KUKA KRL program: EPS_2_251112_SAMH03_A_20250918124115.src

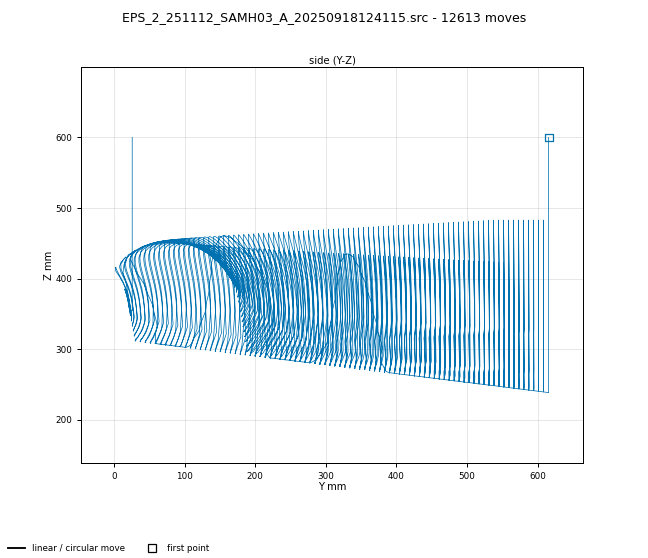
[picture p0: tool path of EPS_2_251112_SAMH03_A_20250918124115.src, 12613 of 12615 moves have a stored position in this frame; points joined in program order, loops and branches not executed]
&ACCESS RVP
&REL 4
&COMMENT QRS 19112012
&PARAM EDITMASK = *
DEF PART()
EXT BAS (BAS_COMMAND :IN,REAL :IN )
INT I
BAS (#INITMOV,0 )

;KUKA QRS Post kuka4.cps  Date:22-06-2017 !

File_ID=2847

QRS_PRE_INIT()

;Init var - Until changes are made in qrs_pre_init
Outlet_Square_prg=0
Inlet_1_Square_prg=0
Inlet_2_Square_prg=0
Inlet_3_Square_prg=0
Inlet_4_Square_prg=0
Inlet_5_Square_prg=0

Outlet_1={X 0.000, Y 541.230, Z 408.000, B 0.000, E1 0.000 }
Inlet_1={X 0.000, Y 545.490, Z 348.000, B 0.000, E1 229.000 }
Outlet_1_type=150
Inlet_1_type=150
;QRS#1=Sidecore dimensions
;QRS#2=150-6" PVC SDR 28
;QRS#3=150-6" PVC SDR 28
;QRS#4=
;QRS#5=
;QRS#6=
;QRS#7=
;QRS#8=
;QRS#9=10-06 PSX
;QRS#10=10-06 PSX
;QRS#11=
;QRS#12=
;QRS#13=
;QRS#14=
;QRS#15=
;QRS#16=1220x127x762 2,5'
;QRS#17=EPS Height
;QRS#18=483
;QRS#19=*
;QRS#20= UPDATED VERSION 22-06-2017
;QRS#21=*
Outlet_Square=070
Inlet_1_Square=070
Inlet_2_Square=0
Inlet_3_Square=0
Inlet_4_Square=0
Inlet_5_Square=0
Mill_Square=1
Outlet_Square_Prg=203
Inlet_1_Square_prg=203

QRS_INIT()

$ADVANCE=5

; T1
PTP {E1 173.598,E2 173.598}
PTP {X 0,Y 615.507,A -85,B 0,C 180,E1 173.598,E2 173.598,E3 0,E4 0,E5 0,E6 0}
QRS_SPEED_INIT()
LIN {X 0,Y 615.507,Z 600,A -85,B 0,C 180,E1 173.598,E2 173.598,E3 0,E4 0,E5 0,E6 0} C_VEL
LIN {X 0,Y 615.507,Z 248.674,A -85,B 0,C 180,E1 173.598,E2 173.598} C_VEL
LIN {X 0,Y 615.507,Z 240.494,A -85,B 0,C 180,E1 173.598,E2 173.598} C_VEL
LIN {X 0,Y 615.49,Z 238.494,A -85,B 0,C 180,E1 173.411,E2 173.411} C_VEL
LIN {X 0,Y 615.479,Z 238.505,A -85,B 0,C 180,E1 170.802,E2 170.802} C_VEL
LIN {X 0,Y 615.478,Z 238.506,A -85,B 0,C 180,E1 168.14,E2 168.14} C_VEL
LIN {X 0,Y 615.488,Z 238.494,A -85,B 0,C 180,E1 165.452,E2 165.452} C_VEL
LIN {X 0,Y 615.482,Z 238.506,A -85,B 0,C 180,E1 162.73,E2 162.73} C_VEL
LIN {X 0,Y 615.471,Z 238.504,A -85,B 0,C 180,E1 159.967,E2 159.967} C_VEL
LIN {X 0,Y 615.483,Z 238.497,A -85,B 0,C 180,E1 157.156,E2 157.156} C_VEL
LIN {X 0,Y 615.486,Z 238.51,A -85,B 0,C 180,E1 154.285,E2 154.285} C_VEL
LIN {X 0,Y 615.486,Z 238.495,A -85,B 0,C 180,E1 151.343,E2 151.343} C_VEL
LIN {X 0,Y 615.488,Z 238.51,A -85,B 0,C 180,E1 148.316,E2 148.316} C_VEL
LIN {X 0,Y 615.471,Z 238.504,A -85,B 0,C 180,E1 145.978,E2 145.978} C_VEL
LIN {X 0,Y 615.477,Z 238.497,A -85,B 0,C 180,E1 143.576,E2 143.576} C_VEL
LIN {X 0,Y 615.483,Z 238.501,A -85,B 0,C 180,E1 140.937,E2 140.937} C_VEL
LIN {X 0,Y 615.491,Z 238.511,A -85,B 0,C 180,E1 138.528,E2 138.528} C_VEL
LIN {X 0,Y 615.467,Z 238.502,A -85,B 0,C 180,E1 135.85,E2 135.85} C_VEL
LIN {X 0,Y 615.489,Z 238.497,A -85,B 0,C 180,E1 133.049,E2 133.049} C_VEL
LIN {X 0,Y 615.49,Z 238.508,A -85,B 0,C 180,E1 130.605,E2 130.605} C_VEL
LIN {X 0,Y 615.468,Z 238.506,A -85,B 0,C 180,E1 128.011,E2 128.011} C_VEL
LIN {X 0,Y 615.465,Z 238.5,A -85,B 0,C 180,E1 125.617,E2 125.617} C_VEL
LIN {X 0,Y 615.483,Z 238.496,A -85,B 0,C 180,E1 123.236,E2 123.236} C_VEL
LIN {X 0,Y 615.485,Z 238.5,A -85,B 0,C 180,E1 120.919,E2 120.919} C_VEL
LIN {X 0,Y 615.498,Z 238.512,A -85,B 0,C 180,E1 118.454,E2 118.454} C_VEL
LIN {X 0,Y 615.462,Z 238.502,A -85,B 0,C 180,E1 115.716,E2 115.716} C_VEL
LIN {X 0,Y 615.465,Z 238.5,A -85,B 0,C 180,E1 113.557,E2 113.557} C_VEL
LIN {X 0,Y 615.489,Z 238.504,A -85,B 0,C 180,E1 110.73,E2 110.73} C_VEL
LIN {X 0,Y 615.462,Z 238.506,A -85,B 0,C 180,E1 107.957,E2 107.957} C_VEL
LIN {X 0,Y 615.484,Z 238.496,A -85,B 0,C 180,E1 105.226,E2 105.226} C_VEL
LIN {X 0,Y 615.487,Z 238.511,A -85,B 0,C 180,E1 102.53,E2 102.53} C_VEL
LIN {X 0,Y 615.454,Z 238.506,A -85,B 0,C 180,E1 99.863,E2 99.863} C_VEL
LIN {X 0,Y 615.48,Z 238.497,A -85,B 0,C 180,E1 97.216,E2 97.216} C_VEL
LIN {X 0,Y 615.491,Z 238.509,A -85,B 0,C 180,E1 94.585,E2 94.585} C_VEL
LIN {X 0,Y 615.459,Z 238.507,A -85,B 0,C 180,E1 91.963,E2 91.963} C_VEL
LIN {X 0,Y 615.462,Z 238.5,A -85,B 0,C 180,E1 89.346,E2 89.346} C_VEL
LIN {X 0,Y 615.493,Z 238.503,A -85,B 0,C 180,E1 86.727,E2 86.727} C_VEL
LIN {X 0,Y 615.466,Z 238.509,A -85,B 0,C 180,E1 84.102,E2 84.102} C_VEL
LIN {X 0,Y 615.454,Z 238.502,A -85,B 0,C 180,E1 81.463,E2 81.463} C_VEL
LIN {X 0,Y 615.495,Z 238.5,A -85,B 0,C 180,E1 78.807,E2 78.807} C_VEL
LIN {X 0,Y 615.463,Z 238.509,A -85,B 0,C 180,E1 76.072,E2 76.072} C_VEL
LIN {X 0,Y 615.448,Z 238.504,A -85,B 0,C 180,E1 73.578,E2 73.578} C_VEL
LIN {X 0,Y 615.495,Z 238.505,A -85,B 0,C 180,E1 70.663,E2 70.663} C_VEL
LIN {X 0,Y 615.449,Z 238.507,A -85,B 0,C 180,E1 67.863,E2 67.863} C_VEL
LIN {X 0,Y 615.445,Z 238.506,A -85,B 0,C 180,E1 65.727,E2 65.727} C_VEL
LIN {X 0,Y 615.442,Z 238.505,A -85,B 0,C 180,E1 63.555,E2 63.555} C_VEL
LIN {X 0,Y 615.495,Z 238.507,A -85,B 0,C 180,E1 60.595,E2 60.595} C_VEL
LIN {X 0,Y 615.482,Z 238.513,A -85,B 0,C 180,E1 58.315,E2 58.315} C_VEL
LIN {X 0,Y 615.48,Z 238.537,A -85,B 0,C 180,E1 56.862,E2 56.862} C_VEL
LIN {X 0,Y 615.452,Z 250.671,A -85,B 0,C 180,E1 54.169,E2 54.169} C_VEL
LIN {X 0,Y 615.422,Z 260.877,A -85,B 0,C 180,E1 51.928,E2 51.928} C_VEL
LIN {X 0,Y 615.463,Z 264.848,A -85,B 0,C 180,E1 51.055,E2 51.055} C_VEL
LIN {X 0,Y 615.43,Z 339.353,A -85,B 0,C 180,E1 50.164,E2 50.164} C_VEL
LIN {X 0,Y 615.423,Z 347.654,A -85,B 0,C 180,E1 49.999,E2 49.999} C_VEL
LIN {X 0,Y 615.423,Z 357.187,A -85,B 0,C 180,E1 49.72,E2 49.72} C_VEL
LIN {X 0,Y 615.442,Z 365.491,A -85,B 0,C 180,E1 49.391,E2 49.391} C_VEL
LIN {X 0,Y 615.489,Z 373.933,A -85,B 0,C 180,E1 48.965,E2 48.965} C_VEL
LIN {X 0,Y 615.484,Z 382.137,A -85,B 0,C 180,E1 48.451,E2 48.451} C_VEL
LIN {X 0,Y 615.498,Z 390.744,A -85,B 0,C 180,E1 47.783,E2 47.783} C_VEL
LIN {X 0,Y 615.495,Z 399.09,A -85,B 0,C 180,E1 46.95,E2 46.95} C_VEL
LIN {X 0,Y 615.492,Z 405.175,A -85,B 0,C 180,E1 46.191,E2 46.191} C_VEL
LIN {X 0,Y 615.495,Z 409.938,A -85,B 0,C 180,E1 45.461,E2 45.461} C_VEL
LIN {X 0,Y 615.495,Z 412.871,A -85,B 0,C 180,E1 44.934,E2 44.934} C_VEL
LIN {X 0,Y 615.493,Z 416.877,A -85,B 0,C 180,E1 43.999,E2 43.999} C_VEL
LIN {X 0,Y 615.491,Z 419.769,A -85,B 0,C 180,E1 43.049,E2 43.049} C_VEL
LIN {X 0,Y 615.494,Z 421.587,A -85,B 0,C 180,E1 42.082,E2 42.082} C_VEL
LIN {X 0,Y 615.494,Z 422.345,A -85,B 0,C 180,E1 41.097,E2 41.097} C_VEL
LIN {X 0,Y 615.491,Z 421.957,A -85,B 0,C 180,E1 40.091,E2 40.091} C_VEL
LIN {X 0,Y 615.493,Z 419.87,A -85,B 0,C 180,E1 38.903,E2 38.903} C_VEL
LIN {X 0,Y 615.49,Z 417.42,A -85,B 0,C 180,E1 38.067,E2 38.067} C_VEL
LIN {X 0,Y 615.494,Z 414.081,A -85,B 0,C 180,E1 37.241,E2 37.241} C_VEL
LIN {X 0,Y 615.496,Z 409.786,A -85,B 0,C 180,E1 36.423,E2 36.423} C_VEL
LIN {X 0,Y 615.495,Z 404.427,A -85,B 0,C 180,E1 35.614,E2 35.614} C_VEL
LIN {X 0,Y 615.496,Z 396.778,A -85,B 0,C 180,E1 34.704,E2 34.704} C_VEL
LIN {X 0,Y 615.496,Z 389.446,A -85,B 0,C 180,E1 34.02,E2 34.02} C_VEL
LIN {X 0,Y 615.478,Z 382.157,A -85,B 0,C 180,E1 33.46,E2 33.46} C_VEL
LIN {X 0,Y 615.497,Z 373.88,A -85,B 0,C 180,E1 32.942,E2 32.942} C_VEL
LIN {X 0,Y 615.477,Z 365.174,A -85,B 0,C 180,E1 32.506,E2 32.506} C_VEL
LIN {X 0,Y 615.449,Z 356.53,A -85,B 0,C 180,E1 32.168,E2 32.168} C_VEL
LIN {X 0,Y 615.442,Z 346.706,A -85,B 0,C 180,E1 31.887,E2 31.887} C_VEL
LIN {X 0,Y 615.446,Z 335.604,A -85,B 0,C 180,E1 31.687,E2 31.687} C_VEL
LIN {X 0,Y 615.496,Z 264.804,A -85,B 0,C 180,E1 30.847,E2 30.847} C_VEL
LIN {X 0,Y 615.464,Z 252.68,A -85,B 0,C 180,E1 28.183,E2 28.183} C_VEL
LIN {X 0,Y 615.493,Z 240.882,A -85,B 0,C 180,E1 25.573,E2 25.573} C_VEL
LIN {X 0,Y 615.483,Z 238.5,A -85,B 0,C 180,E1 24.991,E2 24.991} C_VEL
LIN {X 0,Y 615.471,Z 238.501,A -85,B 0,C 180,E1 22.136,E2 22.136} C_VEL
LIN {X 0,Y 615.488,Z 238.509,A -85,B 0,C 180,E1 19.337,E2 19.337} C_VEL
LIN {X 0,Y 615.483,Z 238.495,A -85,B 0,C 180,E1 16.434,E2 16.434} C_VEL
LIN {X 0,Y 615.476,Z 238.505,A -85,B 0,C 180,E1 13.874,E2 13.874} C_VEL
LIN {X 0,Y 615.482,Z 238.506,A -85,B 0,C 180,E1 11.193,E2 11.193} C_VEL
LIN {X 0,Y 615.489,Z 238.494,A -85,B 0,C 180,E1 8.536,E2 8.536} C_VEL
LIN {X 0,Y 615.477,Z 238.505,A -85,B 0,C 180,E1 5.898,E2 5.898} C_VEL
LIN {X 0,Y 615.484,Z 238.508,A -85,B 0,C 180,E1 3.272,E2 3.272} C_VEL
LIN {X 0,Y 615.482,Z 238.496,A -85,B 0,C 180,E1 0.654,E2 0.654} C_VEL
LIN {X 0,Y 615.478,Z 238.501,A -85,B 0,C 180,E1 -1.964,E2 -1.964} C_VEL
LIN {X 0,Y 615.492,Z 238.511,A -85,B 0,C 180,E1 -4.585,E2 -4.585} C_VEL
LIN {X 0,Y 615.478,Z 238.498,A -85,B 0,C 180,E1 -7.216,E2 -7.216} C_VEL
LIN {X 0,Y 615.48,Z 238.499,A -85,B 0,C 180,E1 -9.863,E2 -9.863} C_VEL
LIN {X 0,Y 615.487,Z 238.514,A -85,B 0,C 180,E1 -12.531,E2 -12.531} C_VEL
LIN {X 0,Y 615.475,Z 238.499,A -85,B 0,C 180,E1 -15.227,E2 -15.227} C_VEL
LIN {X 0,Y 615.482,Z 238.5,A -85,B 0,C 180,E1 -17.957,E2 -17.957} C_VEL
LIN {X 0,Y 615.478,Z 238.509,A -85,B 0,C 180,E1 -20.731,E2 -20.731} C_VEL
LIN {X 0,Y 615.483,Z 238.495,A -85,B 0,C 180,E1 -23.557,E2 -23.557} C_VEL
LIN {X 0,Y 615.49,Z 238.513,A -85,B 0,C 180,E1 -26.444,E2 -26.444} C_VEL
LIN {X 0,Y 615.48,Z 238.511,A -85,B 0,C 180,E1 -28.659,E2 -28.659} C_VEL
LIN {X 0,Y 615.467,Z 238.502,A -85,B 0,C 180,E1 -31.085,E2 -31.085} C_VEL
LIN {X 0,Y 615.482,Z 238.496,A -85,B 0,C 180,E1 -33.535,E2 -33.535} C_VEL
LIN {X 0,Y 615.484,Z 238.514,A -85,B 0,C 180,E1 -36.425,E2 -36.425} C_VEL
LIN {X 0,Y 615.464,Z 238.503,A -85,B 0,C 180,E1 -39.061,E2 -39.061} C_VEL
LIN {X 0,Y 615.477,Z 238.497,A -85,B 0,C 180,E1 -41.475,E2 -41.475} C_VEL
LIN {X 0,Y 615.486,Z 238.504,A -85,B 0,C 180,E1 -44.15,E2 -44.15} C_VEL
LIN {X 0,Y 615.465,Z 238.505,A -85,B 0,C 180,E1 -46.955,E2 -46.955} C_VEL
LIN {X 0,Y 615.468,Z 238.499,A -85,B 0,C 180,E1 -49.393,E2 -49.393} C_VEL
LIN {X 0,Y 615.491,Z 238.499,A -85,B 0,C 180,E1 -51.988,E2 -51.988} C_VEL
LIN {X 0,Y 615.495,Z 238.51,A -85,B 0,C 180,E1 -54.386,E2 -54.386} C_VEL
LIN {X 0,Y 615.473,Z 238.509,A -85,B 0,C 180,E1 -56.764,E2 -56.764} C_VEL
LIN {X 0,Y 615.458,Z 238.505,A -85,B 0,C 180,E1 -59.08,E2 -59.08} C_VEL
LIN {X 0,Y 615.471,Z 238.498,A -85,B 0,C 180,E1 -61.553,E2 -61.553} C_VEL
LIN {X 0,Y 615.497,Z 238.511,A -85,B 0,C 180,E1 -64.429,E2 -64.429} C_VEL
LIN {X 0,Y 615.452,Z 238.505,A -85,B 0,C 180,E1 -67.155,E2 -67.155} C_VEL
LIN {X 0,Y 615.49,Z 238.596,A -85,B 0,C 180,E1 -67.839,E2 -67.839} C_VEL
LIN {X 0,Y 615.444,Z 257.739,A -85,B 0,C 180,E1 -70.661,E2 -70.661} C_VEL
LIN {X 0,Y 615.476,Z 276.68,A -85,B 0,C 180,E1 -73.414,E2 -73.414} C_VEL
LIN {X 0,Y 615.478,Z 296.787,A -85,B 0,C 180,E1 -76.294,E2 -76.294} C_VEL
LIN {X 0,Y 615.469,Z 315.645,A -85,B 0,C 180,E1 -78.966,E2 -78.966} C_VEL
LIN {X 0,Y 615.49,Z 322.035,A -85,B 0,C 180,E1 -79.868,E2 -79.868} C_VEL
LIN {X 0,Y 615.447,Z 399.978,A -85,B 0,C 180,E1 -80.801,E2 -80.801} C_VEL
LIN {X 0,Y 615.437,Z 409.726,A -85,B 0,C 180,E1 -81.008,E2 -81.008} C_VEL
LIN {X 0,Y 615.439,Z 420.178,A -85,B 0,C 180,E1 -81.339,E2 -81.339} C_VEL
LIN {X 0,Y 615.473,Z 430.438,A -85,B 0,C 180,E1 -81.794,E2 -81.794} C_VEL
LIN {X 0,Y 615.478,Z 440.206,A -85,B 0,C 180,E1 -82.372,E2 -82.372} C_VEL
LIN {X 0,Y 615.493,Z 447.938,A -85,B 0,C 180,E1 -82.942,E2 -82.942} C_VEL
LIN {X 0,Y 615.498,Z 455.337,A -85,B 0,C 180,E1 -83.608,E2 -83.608} C_VEL
LIN {X 0,Y 615.498,Z 462.739,A -85,B 0,C 180,E1 -84.431,E2 -84.431} C_VEL
LIN {X 0,Y 615.497,Z 468.534,A -85,B 0,C 180,E1 -85.252,E2 -85.252} C_VEL
LIN {X 0,Y 615.496,Z 473.101,A -85,B 0,C 180,E1 -86.072,E2 -86.072} C_VEL
LIN {X 0,Y 615.493,Z 476.069,A -85,B 0,C 180,E1 -86.727,E2 -86.727} C_VEL
LIN {X 0,Y 615.494,Z 478.357,A -85,B 0,C 180,E1 -87.382,E2 -87.382} C_VEL
LIN {X 0,Y 615.499,Z 480.085,A -85,B 0,C 180,E1 -88.037,E2 -88.037} C_VEL
LIN {X 0,Y 615.493,Z 481.33,A -85,B 0,C 180,E1 -88.692,E2 -88.692} C_VEL
LIN {X 0,Y 615.491,Z 482.104,A -85,B 0,C 180,E1 -89.346,E2 -89.346} C_VEL
LIN {X 0,Y 615.491,Z 482.389,A -85,B 0,C 180,E1 -90,E2 -90} C_VEL
LIN {X 0,Y 615.491,Z 482.104,A -85,B 0,C 180,E1 -90.654,E2 -90.654} C_VEL
LIN {X 0,Y 615.493,Z 481.33,A -85,B 0,C 180,E1 -91.309,E2 -91.309} C_VEL
LIN {X 0,Y 615.499,Z 480.085,A -85,B 0,C 180,E1 -91.963,E2 -91.963} C_VEL
LIN {X 0,Y 615.488,Z 477.22,A -85,B 0,C 180,E1 -92.945,E2 -92.945} C_VEL
LIN {X 0,Y 615.493,Z 474.602,A -85,B 0,C 180,E1 -93.601,E2 -93.601} C_VEL
LIN {X 0,Y 615.495,Z 469.482,A -85,B 0,C 180,E1 -94.585,E2 -94.585} C_VEL
LIN {X 0,Y 615.495,Z 463.968,A -85,B 0,C 180,E1 -95.405,E2 -95.405} C_VEL
LIN {X 0,Y 615.498,Z 457.017,A -85,B 0,C 180,E1 -96.227,E2 -96.227} C_VEL
LIN {X 0,Y 615.495,Z 449.859,A -85,B 0,C 180,E1 -96.901,E2 -96.901} C_VEL
LIN {X 0,Y 615.477,Z 442.624,A -85,B 0,C 180,E1 -97.463,E2 -97.463} C_VEL
LIN {X 0,Y 615.495,Z 434.868,A -85,B 0,C 180,E1 -97.958,E2 -97.958} C_VEL
LIN {X 0,Y 615.456,Z 426.924,A -85,B 0,C 180,E1 -98.372,E2 -98.372} C_VEL
LIN {X 0,Y 615.436,Z 417.772,A -85,B 0,C 180,E1 -98.744,E2 -98.744} C_VEL
LIN {X 0,Y 615.438,Z 409.713,A -85,B 0,C 180,E1 -98.992,E2 -98.992} C_VEL
LIN {X 0,Y 615.447,Z 399.958,A -85,B 0,C 180,E1 -99.199,E2 -99.199} C_VEL
LIN {X 0,Y 615.49,Z 322.033,A -85,B 0,C 180,E1 -100.132,E2 -100.132} C_VEL
LIN {X 0,Y 615.485,Z 302.697,A -85,B 0,C 180,E1 -102.865,E2 -102.865} C_VEL
LIN {X 0,Y 615.46,Z 283.779,A -85,B 0,C 180,E1 -105.566,E2 -105.566} C_VEL
LIN {X 0,Y 615.461,Z 263.931,A -85,B 0,C 180,E1 -108.434,E2 -108.434} C_VEL
LIN {X 0,Y 615.455,Z 247.068,A -85,B 0,C 180,E1 -110.907,E2 -110.907} C_VEL
LIN {X 0,Y 615.487,Z 238.497,A -85,B 0,C 180,E1 -112.187,E2 -112.187} C_VEL
LIN {X 0,Y 615.458,Z 238.506,A -85,B 0,C 180,E1 -114.993,E2 -114.993} C_VEL
LIN {X 0,Y 615.491,Z 238.501,A -85,B 0,C 180,E1 -117.914,E2 -117.914} C_VEL
LIN {X 0,Y 615.499,Z 238.494,A -85,B 0,C 180,E1 -120.159,E2 -120.159} C_VEL
LIN {X 0,Y 615.473,Z 238.498,A -85,B 0,C 180,E1 -122.458,E2 -122.458} C_VEL
LIN {X 0,Y 615.458,Z 238.503,A -85,B 0,C 180,E1 -124.816,E2 -124.816} C_VEL
LIN {X 0,Y 615.473,Z 238.509,A -85,B 0,C 180,E1 -127.243,E2 -127.243} C_VEL
LIN {X 0,Y 615.493,Z 238.497,A -85,B 0,C 180,E1 -130.089,E2 -130.089} C_VEL
LIN {X 0,Y 615.487,Z 238.495,A -85,B 0,C 180,E1 -132.352,E2 -132.352} C_VEL
LIN {X 0,Y 615.465,Z 238.506,A -85,B 0,C 180,E1 -135.07,E2 -135.07} C_VEL
LIN {X 0,Y 615.486,Z 238.502,A -85,B 0,C 180,E1 -137.919,E2 -137.919} C_VEL
LIN {X 0,Y 615.498,Z 238.493,A -85,B 0,C 180,E1 -140.25,E2 -140.25} C_VEL
LIN {X 0,Y 615.467,Z 238.505,A -85,B 0,C 180,E1 -143.065,E2 -143.065} C_VEL
LIN {X 0,Y 615.475,Z 238.51,A -85,B 0,C 180,E1 -145.3,E2 -145.3} C_VEL
LIN {X 0,Y 615.492,Z 238.509,A -85,B 0,C 180,E1 -147.667,E2 -147.667} C_VEL
LIN {X 0,Y 615.477,Z 238.497,A -85,B 0,C 180,E1 -150.593,E2 -150.593} C_VEL
LIN {X 0,Y 615.467,Z 238.503,A -85,B 0,C 180,E1 -152.957,E2 -152.957} C_VEL
LIN {X 0,Y 615.489,Z 238.508,A -85,B 0,C 180,E1 -155.728,E2 -155.728} C_VEL
LIN {X 0,Y 615.483,Z 238.495,A -85,B 0,C 180,E1 -158.568,E2 -158.568} C_VEL
LIN {X 0,Y 615.487,Z 238.51,A -85,B 0,C 180,E1 -161.393,E2 -161.393} C_VEL
LIN {X 0,Y 615.484,Z 238.499,A -85,B 0,C 180,E1 -164.094,E2 -164.094} C_VEL
LIN {X 0,Y 615.474,Z 238.499,A -85,B 0,C 180,E1 -166.798,E2 -166.798} C_VEL
LIN {X 0,Y 615.493,Z 238.512,A -85,B 0,C 180,E1 -169.473,E2 -169.473} C_VEL
LIN {X 0,Y 615.482,Z 238.499,A -85,B 0,C 180,E1 -172.124,E2 -172.124} C_VEL
LIN {X 0,Y 615.479,Z 238.497,A -85,B 0,C 180,E1 -174.758,E2 -174.758} C_VEL
LIN {X 0,Y 615.487,Z 238.509,A -85,B 0,C 180,E1 -177.382,E2 -177.382} C_VEL
LIN {X 0,Y 615.479,Z 238.503,A -85,B 0,C 180,E1 -179.999,E2 -179.999} C_VEL
LIN {X 0,Y 615.491,Z 238.493,A -85,B 0,C 180,E1 -182.617,E2 -182.617} C_VEL
LIN {X 0,Y 615.475,Z 238.507,A -85,B 0,C 180,E1 -185.241,E2 -185.241} C_VEL
LIN {X 0,Y 615.49,Z 238.494,A -85,B 0,C 180,E1 -186.589,E2 -186.589} C_VEL
LIN {X 0,Y 614.807,Z 238.652,A -85,B 0,C 180,E1 -187.135,E2 -187.135} C_VEL
LIN {X 0,Y 611.967,Z 239.065,A -85,B 0,C 180,E1 -188.021,E2 -188.021} C_VEL
LIN {X 0,Y 609.575,Z 239.378,A -85,B 0,C 180,E1 -188.733,E2 -188.733} C_VEL
LIN {X 0,Y 608.541,Z 239.496,A -85,B 0,C 180,E1 -189.283,E2 -189.283} C_VEL
LIN {X 0,Y 608.452,Z 239.505,A -85,B 0,C 180,E1 -189.469,E2 -189.469} C_VEL
LIN {X 0,Y 608.456,Z 239.503,A -85,B 0,C 180,E1 -191.999,E2 -191.999} C_VEL
LIN {X 0,Y 608.473,Z 239.497,A -85,B 0,C 180,E1 -194.72,E2 -194.72} C_VEL
LIN {X 0,Y 608.446,Z 239.51,A -85,B 0,C 180,E1 -197.476,E2 -197.476} C_VEL
LIN {X 0,Y 608.454,Z 239.5,A -85,B 0,C 180,E1 -200.274,E2 -200.274} C_VEL
LIN {X 0,Y 608.448,Z 239.5,A -85,B 0,C 180,E1 -202.476,E2 -202.476} C_VEL
LIN {X 0,Y 608.454,Z 239.506,A -85,B 0,C 180,E1 -205.3,E2 -205.3} C_VEL
LIN {X 0,Y 608.441,Z 239.512,A -85,B 0,C 180,E1 -207.517,E2 -207.517} C_VEL
LIN {X 0,Y 608.458,Z 239.503,A -85,B 0,C 180,E1 -209.972,E2 -209.972} C_VEL
LIN {X 0,Y 608.455,Z 239.499,A -85,B 0,C 180,E1 -212.523,E2 -212.523} C_VEL
LIN {X 0,Y 608.448,Z 239.506,A -85,B 0,C 180,E1 -215.276,E2 -215.276} C_VEL
LIN {X 0,Y 608.458,Z 239.506,A -85,B 0,C 180,E1 -217.746,E2 -217.746} C_VEL
LIN {X 0,Y 608.44,Z 239.502,A -85,B 0,C 180,E1 -220.329,E2 -220.329} C_VEL
LIN {X 0,Y 608.471,Z 239.504,A -85,B 0,C 180,E1 -223.31,E2 -223.31} C_VEL
LIN {X 0,Y 608.458,Z 239.501,A -85,B 0,C 180,E1 -226.13,E2 -226.13} C_VEL
LIN {X 0,Y 608.455,Z 239.5,A -85,B 0,C 180,E1 -228.824,E2 -228.824} C_VEL
LIN {X 0,Y 608.463,Z 239.506,A -85,B 0,C 180,E1 -231.412,E2 -231.412} C_VEL
LIN {X 0,Y 608.434,Z 239.506,A -85,B 0,C 180,E1 -233.954,E2 -233.954} C_VEL
LIN {X 0,Y 608.437,Z 239.502,A -85,B 0,C 180,E1 -236.328,E2 -236.328} C_VEL
LIN {X 0,Y 608.47,Z 239.498,A -85,B 0,C 180,E1 -238.727,E2 -238.727} C_VEL
LIN {X 0,Y 608.451,Z 239.508,A -85,B 0,C 180,E1 -241.734,E2 -241.734} C_VEL
LIN {X 0,Y 608.451,Z 239.501,A -85,B 0,C 180,E1 -244.281,E2 -244.281} C_VEL
LIN {X 0,Y 608.443,Z 239.502,A -85,B 0,C 180,E1 -246.876,E2 -246.876} C_VEL
LIN {X 0,Y 608.455,Z 239.507,A -85,B 0,C 180,E1 -249.726,E2 -249.726} C_VEL
LIN {X 0,Y 608.435,Z 239.508,A -85,B 0,C 180,E1 -251.828,E2 -251.828} C_VEL
LIN {X 0,Y 608.446,Z 239.505,A -85,B 0,C 180,E1 -253.906,E2 -253.906} C_VEL
LIN {X 0,Y 608.443,Z 239.505,A -85,B 0,C 180,E1 -255.988,E2 -255.988} C_VEL
LIN {X 0,Y 608.469,Z 239.498,A -85,B 0,C 180,E1 -258.676,E2 -258.676} C_VEL
LIN {X 0,Y 608.457,Z 239.506,A -85,B 0,C 180,E1 -261.364,E2 -261.364} C_VEL
LIN {X 0,Y 608.436,Z 239.505,A -85,B 0,C 180,E1 -264.033,E2 -264.033} C_VEL
LIN {X 0,Y 608.465,Z 239.498,A -85,B 0,C 180,E1 -266.689,E2 -266.689} C_VEL
LIN {X 0,Y 608.482,Z 239.502,A -85,B 0,C 180,E1 -269.338,E2 -269.338} C_VEL
LIN {X 0,Y 608.432,Z 239.506,A -85,B 0,C 180,E1 -271.986,E2 -271.986} C_VEL
LIN {X 0,Y 608.433,Z 239.506,A -85,B 0,C 180,E1 -273.974,E2 -273.974} C_VEL
LIN {X 0,Y 608.429,Z 239.503,A -85,B 0,C 180,E1 -276.633,E2 -276.633} C_VEL
LIN {X 0,Y 608.471,Z 239.503,A -85,B 0,C 180,E1 -279.305,E2 -279.305} C_VEL
LIN {X 0,Y 608.442,Z 239.505,A -85,B 0,C 180,E1 -282,E2 -282} C_VEL
LIN {X 0,Y 608.453,Z 239.5,A -85,B 0,C 180,E1 -284.721,E2 -284.721} C_VEL
LIN {X 0,Y 608.449,Z 239.509,A -85,B 0,C 180,E1 -287.476,E2 -287.476} C_VEL
LIN {X 0,Y 608.43,Z 239.503,A -85,B 0,C 180,E1 -290.275,E2 -290.275} C_VEL
LIN {X 0,Y 608.431,Z 239.502,A -85,B 0,C 180,E1 -292.473,E2 -292.473} C_VEL
LIN {X 0,Y 608.453,Z 239.505,A -85,B 0,C 180,E1 -295.3,E2 -295.3} C_VEL
LIN {X 0,Y 608.439,Z 239.511,A -85,B 0,C 180,E1 -297.518,E2 -297.518} C_VEL
LIN {X 0,Y 608.429,Z 239.507,A -85,B 0,C 180,E1 -299.967,E2 -299.967} C_VEL
LIN {X 0,Y 608.42,Z 239.504,A -85,B 0,C 180,E1 -302.518,E2 -302.518} C_VEL
LIN {X 0,Y 608.468,Z 239.719,A -85,B 0,C 180,E1 -303.174,E2 -303.174} C_VEL
LIN {X 0,Y 608.391,Z 252.562,A -85,B 0,C 180,E1 -306.04,E2 -306.04} C_VEL
LIN {X 0,Y 608.39,Z 262.483,A -85,B 0,C 180,E1 -308.233,E2 -308.233} C_VEL
LIN {X 0,Y 608.419,Z 265.192,A -85,B 0,C 180,E1 -308.829,E2 -308.829} C_VEL
LIN {X 0,Y 608.433,Z 340.315,A -85,B 0,C 180,E1 -309.737,E2 -309.737} C_VEL
LIN {X 0,Y 608.425,Z 350.261,A -85,B 0,C 180,E1 -309.953,E2 -309.953} C_VEL
LIN {X 0,Y 608.418,Z 361.668,A -85,B 0,C 180,E1 -310.327,E2 -310.327} C_VEL
LIN {X 0,Y 608.478,Z 372.532,A -85,B 0,C 180,E1 -310.844,E2 -310.844} C_VEL
LIN {X 0,Y 608.47,Z 380.777,A -85,B 0,C 180,E1 -311.345,E2 -311.345} C_VEL
LIN {X 0,Y 608.447,Z 387.854,A -85,B 0,C 180,E1 -311.867,E2 -311.867} C_VEL
LIN {X 0,Y 608.449,Z 394.437,A -85,B 0,C 180,E1 -312.45,E2 -312.45} C_VEL
LIN {X 0,Y 608.45,Z 400.823,A -85,B 0,C 180,E1 -313.132,E2 -313.132} C_VEL
LIN {X 0,Y 608.432,Z 406.518,A -85,B 0,C 180,E1 -313.871,E2 -313.871} C_VEL
LIN {X 0,Y 608.429,Z 412.234,A -85,B 0,C 180,E1 -314.797,E2 -314.797} C_VEL
LIN {X 0,Y 608.446,Z 416.628,A -85,B 0,C 180,E1 -315.736,E2 -315.736} C_VEL
LIN {X 0,Y 608.429,Z 419.796,A -85,B 0,C 180,E1 -316.694,E2 -316.694} C_VEL
LIN {X 0,Y 608.422,Z 422.239,A -85,B 0,C 180,E1 -317.937,E2 -317.937} C_VEL
LIN {X 0,Y 608.429,Z 422.92,A -85,B 0,C 180,E1 -318.823,E2 -318.823} C_VEL
LIN {X 0,Y 608.438,Z 422.718,A -85,B 0,C 180,E1 -319.697,E2 -319.697} C_VEL
LIN {X 0,Y 608.446,Z 421.437,A -85,B 0,C 180,E1 -320.704,E2 -320.704} C_VEL
LIN {X 0,Y 608.42,Z 418.688,A -85,B 0,C 180,E1 -321.764,E2 -321.764} C_VEL
LIN {X 0,Y 608.423,Z 415.661,A -85,B 0,C 180,E1 -322.575,E2 -322.575} C_VEL
LIN {X 0,Y 608.455,Z 411.045,A -85,B 0,C 180,E1 -323.499,E2 -323.499} C_VEL
LIN {X 0,Y 608.443,Z 407.033,A -85,B 0,C 180,E1 -324.146,E2 -324.146} C_VEL
LIN {X 0,Y 608.463,Z 400.994,A -85,B 0,C 180,E1 -324.938,E2 -324.938} C_VEL
LIN {X 0,Y 608.453,Z 394.527,A -85,B 0,C 180,E1 -325.631,E2 -325.631} C_VEL
LIN {X 0,Y 608.447,Z 386.559,A -85,B 0,C 180,E1 -326.329,E2 -326.329} C_VEL
LIN {X 0,Y 608.478,Z 376.473,A -85,B 0,C 180,E1 -327.024,E2 -327.024} C_VEL
LIN {X 0,Y 608.481,Z 366.615,A -85,B 0,C 180,E1 -327.542,E2 -327.542} C_VEL
LIN {X 0,Y 608.452,Z 357.646,A -85,B 0,C 180,E1 -327.906,E2 -327.906} C_VEL
LIN {X 0,Y 608.452,Z 348.309,A -85,B 0,C 180,E1 -328.186,E2 -328.186} C_VEL
LIN {X 0,Y 608.459,Z 339.339,A -85,B 0,C 180,E1 -328.369,E2 -328.369} C_VEL
LIN {X 0,Y 608.463,Z 265.177,A -85,B 0,C 180,E1 -329.264,E2 -329.264} C_VEL
LIN {X 0,Y 608.435,Z 252.294,A -85,B 0,C 180,E1 -332.108,E2 -332.108} C_VEL
LIN {X 0,Y 608.472,Z 239.5,A -85,B 0,C 180,E1 -334.975,E2 -334.975} C_VEL
LIN {X 0,Y 608.463,Z 239.498,A -85,B 0,C 180,E1 -337.595,E2 -337.595} C_VEL
LIN {X 0,Y 608.447,Z 239.51,A -85,B 0,C 180,E1 -340.43,E2 -340.43} C_VEL
LIN {X 0,Y 608.467,Z 239.498,A -85,B 0,C 180,E1 -343.467,E2 -343.467} C_VEL
LIN {X 0,Y 608.461,Z 239.501,A -85,B 0,C 180,E1 -345.981,E2 -345.981} C_VEL
LIN {X 0,Y 608.469,Z 239.505,A -85,B 0,C 180,E1 -348.677,E2 -348.677} C_VEL
LIN {X 0,Y 608.457,Z 239.499,A -85,B 0,C 180,E1 -351.365,E2 -351.365} C_VEL
LIN {X 0,Y 608.452,Z 239.503,A -85,B 0,C 180,E1 -354.034,E2 -354.034} C_VEL
LIN {X 0,Y 608.475,Z 239.504,A -85,B 0,C 180,E1 -356.69,E2 -356.69} C_VEL
LIN {X 0,Y 608.475,Z 239.497,A -85,B 0,C 180,E1 -359.339,E2 -359.339} C_VEL
LIN {X 0,Y 608.448,Z 239.503,A -85,B 0,C 180,E1 -361.986,E2 -361.986} C_VEL
LIN {X 0,Y 608.459,Z 239.507,A -85,B 0,C 180,E1 -364.638,E2 -364.638} C_VEL
LIN {X 0,Y 608.474,Z 239.497,A -85,B 0,C 180,E1 -367.3,E2 -367.3} C_VEL
LIN {X 0,Y 608.452,Z 239.502,A -85,B 0,C 180,E1 -369.978,E2 -369.978} C_VEL
LIN {X 0,Y 608.473,Z 239.505,A -85,B 0,C 180,E1 -372.677,E2 -372.677} C_VEL
LIN {X 0,Y 608.462,Z 239.498,A -85,B 0,C 180,E1 -375.407,E2 -375.407} C_VEL
LIN {X 0,Y 608.448,Z 239.505,A -85,B 0,C 180,E1 -378.172,E2 -378.172} C_VEL
LIN {X 0,Y 608.45,Z 239.503,A -85,B 0,C 180,E1 -380.982,E2 -380.982} C_VEL
LIN {X 0,Y 608.442,Z 239.502,A -85,B 0,C 180,E1 -383.125,E2 -383.125} C_VEL
LIN {X 0,Y 608.476,Z 239.497,A -85,B 0,C 180,E1 -385.724,E2 -385.724} C_VEL
LIN {X 0,Y 608.472,Z 239.506,A -85,B 0,C 180,E1 -388.622,E2 -388.622} C_VEL
LIN {X 0,Y 608.452,Z 239.5,A -85,B 0,C 180,E1 -391.318,E2 -391.318} C_VEL
LIN {X 0,Y 608.469,Z 239.498,A -85,B 0,C 180,E1 -393.736,E2 -393.736} C_VEL
LIN {X 0,Y 608.473,Z 239.501,A -85,B 0,C 180,E1 -396.091,E2 -396.091} C_VEL
LIN {X 0,Y 608.458,Z 239.508,A -85,B 0,C 180,E1 -398.589,E2 -398.589} C_VEL
LIN {X 0,Y 608.448,Z 239.5,A -85,B 0,C 180,E1 -401.342,E2 -401.342} C_VEL
LIN {X 0,Y 608.453,Z 239.506,A -85,B 0,C 180,E1 -404.265,E2 -404.265} C_VEL
LIN {X 0,Y 608.434,Z 239.504,A -85,B 0,C 180,E1 -407.04,E2 -407.04} C_VEL
LIN {X 0,Y 608.448,Z 239.501,A -85,B 0,C 180,E1 -409.698,E2 -409.698} C_VEL
LIN {X 0,Y 608.469,Z 239.504,A -85,B 0,C 180,E1 -412.255,E2 -412.255} C_VEL
LIN {X 0,Y 608.437,Z 239.508,A -85,B 0,C 180,E1 -414.723,E2 -414.723} C_VEL
LIN {X 0,Y 608.446,Z 239.502,A -85,B 0,C 180,E1 -417.121,E2 -417.121} C_VEL
LIN {X 0,Y 608.471,Z 239.501,A -85,B 0,C 180,E1 -420.028,E2 -420.028} C_VEL
LIN {X 0,Y 608.463,Z 239.504,A -85,B 0,C 180,E1 -422.796,E2 -422.796} C_VEL
LIN {X 0,Y 608.441,Z 239.501,A -85,B 0,C 180,E1 -425.429,E2 -425.429} C_VEL
LIN {X 0,Y 608.481,Z 239.663,A -85,B 0,C 180,E1 -427.73,E2 -427.73} C_VEL
LIN {X 0,Y 608.509,Z 256.575,A -85,B 0,C 180,E1 -430.256,E2 -430.256} C_VEL
LIN {X 0,Y 608.446,Z 274.378,A -85,B 0,C 180,E1 -432.87,E2 -432.87} C_VEL
LIN {X 0,Y 608.473,Z 292.18,A -85,B 0,C 180,E1 -435.451,E2 -435.451} C_VEL
LIN {X 0,Y 608.47,Z 311.169,A -85,B 0,C 180,E1 -438.17,E2 -438.17} C_VEL
LIN {X 0,Y 608.463,Z 322.296,A -85,B 0,C 180,E1 -439.75,E2 -439.75} C_VEL
LIN {X 0,Y 608.474,Z 400.465,A -85,B 0,C 180,E1 -440.695,E2 -440.695} C_VEL
LIN {X 0,Y 608.439,Z 410.088,A -85,B 0,C 180,E1 -440.904,E2 -440.904} C_VEL
LIN {X 0,Y 608.428,Z 421.626,A -85,B 0,C 180,E1 -441.28,E2 -441.28} C_VEL
LIN {X 0,Y 608.472,Z 432.238,A -85,B 0,C 180,E1 -441.783,E2 -441.783} C_VEL
LIN {X 0,Y 608.458,Z 440.546,A -85,B 0,C 180,E1 -442.284,E2 -442.284} C_VEL
LIN {X 0,Y 608.459,Z 448.404,A -85,B 0,C 180,E1 -442.868,E2 -442.868} C_VEL
LIN {X 0,Y 608.466,Z 455.358,A -85,B 0,C 180,E1 -443.496,E2 -443.496} C_VEL
LIN {X 0,Y 608.469,Z 463.193,A -85,B 0,C 180,E1 -444.366,E2 -444.366} C_VEL
LIN {X 0,Y 608.448,Z 469.028,A -85,B 0,C 180,E1 -445.197,E2 -445.197} C_VEL
LIN {X 0,Y 608.434,Z 473.632,A -85,B 0,C 180,E1 -446.026,E2 -446.026} C_VEL
LIN {X 0,Y 608.425,Z 476.622,A -85,B 0,C 180,E1 -446.689,E2 -446.689} C_VEL
LIN {X 0,Y 608.423,Z 478.932,A -85,B 0,C 180,E1 -447.352,E2 -447.352} C_VEL
LIN {X 0,Y 608.444,Z 480.679,A -85,B 0,C 180,E1 -448.014,E2 -448.014} C_VEL
LIN {X 0,Y 608.446,Z 481.934,A -85,B 0,C 180,E1 -448.676,E2 -448.676} C_VEL
LIN {X 0,Y 608.434,Z 482.714,A -85,B 0,C 180,E1 -449.338,E2 -449.338} C_VEL
LIN {X 0,Y 608.431,Z 483,A -85,B 0,C 180,E1 -450,E2 -450} C_VEL
LIN {X 0,Y 608.434,Z 482.714,A -85,B 0,C 180,E1 -450.662,E2 -450.662} C_VEL
LIN {X 0,Y 608.445,Z 481.933,A -85,B 0,C 180,E1 -451.324,E2 -451.324} C_VEL
LIN {X 0,Y 608.444,Z 480.678,A -85,B 0,C 180,E1 -451.986,E2 -451.986} C_VEL
LIN {X 0,Y 608.444,Z 477.785,A -85,B 0,C 180,E1 -452.98,E2 -452.98} C_VEL
LIN {X 0,Y 608.447,Z 475.146,A -85,B 0,C 180,E1 -453.642,E2 -453.642} C_VEL
LIN {X 0,Y 608.431,Z 469.984,A -85,B 0,C 180,E1 -454.638,E2 -454.638} C_VEL
LIN {X 0,Y 608.46,Z 464.429,A -85,B 0,C 180,E1 -455.468,E2 -455.468} C_VEL
LIN {X 0,Y 608.455,Z 456.67,A -85,B 0,C 180,E1 -456.376,E2 -456.376} C_VEL
LIN {X 0,Y 608.452,Z 449.414,A -85,B 0,C 180,E1 -457.049,E2 -457.049} C_VEL
LIN {X 0,Y 608.459,Z 441.76,A -85,B 0,C 180,E1 -457.633,E2 -457.633} C_VEL
LIN {X 0,Y 608.483,Z 433.719,A -85,B 0,C 180,E1 -458.134,E2 -458.134} C_VEL
LIN {X 0,Y 608.452,Z 425.389,A -85,B 0,C 180,E1 -458.552,E2 -458.552} C_VEL
LIN {X 0,Y 608.433,Z 416.888,A -85,B 0,C 180,E1 -458.887,E2 -458.887} C_VEL
LIN {X 0,Y 608.439,Z 407.585,A -85,B 0,C 180,E1 -459.16,E2 -459.16} C_VEL
LIN {X 0,Y 608.482,Z 396.548,A -85,B 0,C 180,E1 -459.368,E2 -459.368} C_VEL
LIN {X 0,Y 608.463,Z 322.293,A -85,B 0,C 180,E1 -460.25,E2 -460.25} C_VEL
LIN {X 0,Y 608.481,Z 301.672,A -85,B 0,C 180,E1 -463.186,E2 -463.186} C_VEL
LIN {X 0,Y 608.489,Z 281.496,A -85,B 0,C 180,E1 -466.093,E2 -466.093} C_VEL
LIN {X 0,Y 608.478,Z 262.507,A -85,B 0,C 180,E1 -468.869,E2 -468.869} C_VEL
LIN {X 0,Y 608.546,Z 244.704,A -85,B 0,C 180,E1 -471.51,E2 -471.51} C_VEL
LIN {X 0,Y 608.447,Z 239.502,A -85,B 0,C 180,E1 -472.317,E2 -472.317} C_VEL
LIN {X 0,Y 608.441,Z 239.501,A -85,B 0,C 180,E1 -474.571,E2 -474.571} C_VEL
LIN {X 0,Y 608.463,Z 239.504,A -85,B 0,C 180,E1 -477.204,E2 -477.204} C_VEL
LIN {X 0,Y 608.471,Z 239.501,A -85,B 0,C 180,E1 -479.972,E2 -479.972} C_VEL
LIN {X 0,Y 608.446,Z 239.502,A -85,B 0,C 180,E1 -482.88,E2 -482.88} C_VEL
LIN {X 0,Y 608.438,Z 239.508,A -85,B 0,C 180,E1 -485.277,E2 -485.277} C_VEL
LIN {X 0,Y 608.468,Z 239.498,A -85,B 0,C 180,E1 -488.24,E2 -488.24} C_VEL
LIN {X 0,Y 608.456,Z 239.507,A -85,B 0,C 180,E1 -491.341,E2 -491.341} C_VEL
LIN {X 0,Y 608.459,Z 239.499,A -85,B 0,C 180,E1 -494.264,E2 -494.264} C_VEL
LIN {X 0,Y 608.432,Z 239.505,A -85,B 0,C 180,E1 -497.038,E2 -497.038} C_VEL
LIN {X 0,Y 608.45,Z 239.508,A -85,B 0,C 180,E1 -499.696,E2 -499.696} C_VEL
LIN {X 0,Y 608.464,Z 239.499,A -85,B 0,C 180,E1 -502.253,E2 -502.253} C_VEL
LIN {X 0,Y 608.439,Z 239.502,A -85,B 0,C 180,E1 -504.722,E2 -504.722} C_VEL
LIN {X 0,Y 608.465,Z 239.508,A -85,B 0,C 180,E1 -507.476,E2 -507.476} C_VEL
LIN {X 0,Y 608.474,Z 239.498,A -85,B 0,C 180,E1 -510.221,E2 -510.221} C_VEL
LIN {X 0,Y 608.464,Z 239.499,A -85,B 0,C 180,E1 -512.794,E2 -512.794} C_VEL
LIN {X 0,Y 608.447,Z 239.509,A -85,B 0,C 180,E1 -515.428,E2 -515.428} C_VEL
LIN {X 0,Y 608.466,Z 239.498,A -85,B 0,C 180,E1 -518.308,E2 -518.308} C_VEL
LIN {X 0,Y 608.451,Z 239.504,A -85,B 0,C 180,E1 -521.13,E2 -521.13} C_VEL
LIN {X 0,Y 608.46,Z 239.503,A -85,B 0,C 180,E1 -523.906,E2 -523.906} C_VEL
LIN {X 0,Y 608.454,Z 239.499,A -85,B 0,C 180,E1 -526.643,E2 -526.643} C_VEL
LIN {X 0,Y 608.464,Z 239.506,A -85,B 0,C 180,E1 -529.35,E2 -529.35} C_VEL
LIN {X 0,Y 608.473,Z 239.5,A -85,B 0,C 180,E1 -532.033,E2 -532.033} C_VEL
LIN {X 0,Y 608.458,Z 239.499,A -85,B 0,C 180,E1 -534.698,E2 -534.698} C_VEL
LIN {X 0,Y 608.477,Z 239.504,A -85,B 0,C 180,E1 -537.351,E2 -537.351} C_VEL
LIN {X 0,Y 608.469,Z 239.501,A -85,B 0,C 180,E1 -539.999,E2 -539.999} C_VEL
LIN {X 0,Y 608.481,Z 239.496,A -85,B 0,C 180,E1 -542.647,E2 -542.647} C_VEL
LIN {X 0,Y 608.455,Z 239.506,A -85,B 0,C 180,E1 -545.301,E2 -545.301} C_VEL
LIN {X 0,Y 608.472,Z 239.501,A -85,B 0,C 180,E1 -547.966,E2 -547.966} C_VEL
LIN {X 0,Y 608.452,Z 239.505,A -85,B 0,C 180,E1 -549.469,E2 -549.469} C_VEL
LIN {X 0,Y 607.773,Z 239.588,A -85,B 0,C 180,E1 -550.022,E2 -550.022} C_VEL
LIN {X 0,Y 604.919,Z 239.941,A -85,B 0,C 180,E1 -550.919,E2 -550.919} C_VEL
LIN {X 0,Y 602.516,Z 240.248,A -85,B 0,C 180,E1 -551.64,E2 -551.64} C_VEL
LIN {X 0,Y 601.488,Z 240.369,A -85,B 0,C 180,E1 -552.197,E2 -552.197} C_VEL
LIN {X 0,Y 601.406,Z 240.378,A -85,B 0,C 180,E1 -552.385,E2 -552.385} C_VEL
LIN {X 0,Y 601.426,Z 240.376,A -85,B 0,C 180,E1 -554.896,E2 -554.896} C_VEL
LIN {X 0,Y 601.427,Z 240.377,A -85,B 0,C 180,E1 -556.985,E2 -556.985} C_VEL
LIN {X 0,Y 601.399,Z 240.384,A -85,B 0,C 180,E1 -559.809,E2 -559.809} C_VEL
LIN {X 0,Y 601.405,Z 240.377,A -85,B 0,C 180,E1 -562.605,E2 -562.605} C_VEL
LIN {X 0,Y 601.399,Z 240.379,A -85,B 0,C 180,E1 -564.878,E2 -564.878} C_VEL
LIN {X 0,Y 601.413,Z 240.382,A -85,B 0,C 180,E1 -567.867,E2 -567.867} C_VEL
LIN {X 0,Y 601.418,Z 240.378,A -85,B 0,C 180,E1 -570.164,E2 -570.164} C_VEL
LIN {X 0,Y 601.417,Z 240.376,A -85,B 0,C 180,E1 -572.716,E2 -572.716} C_VEL
LIN {X 0,Y 601.415,Z 240.38,A -85,B 0,C 180,E1 -575.116,E2 -575.116} C_VEL
LIN {X 0,Y 601.425,Z 240.383,A -85,B 0,C 180,E1 -577.419,E2 -577.419} C_VEL
LIN {X 0,Y 601.401,Z 240.382,A -85,B 0,C 180,E1 -579.995,E2 -579.995} C_VEL
LIN {X 0,Y 601.403,Z 240.378,A -85,B 0,C 180,E1 -582.67,E2 -582.67} C_VEL
LIN {X 0,Y 601.415,Z 240.386,A -85,B 0,C 180,E1 -585.482,E2 -585.482} C_VEL
LIN {X 0,Y 601.416,Z 240.376,A -85,B 0,C 180,E1 -588.406,E2 -588.406} C_VEL
LIN {X 0,Y 601.429,Z 240.376,A -85,B 0,C 180,E1 -590.876,E2 -590.876} C_VEL
LIN {X 0,Y 601.413,Z 240.384,A -85,B 0,C 180,E1 -593.736,E2 -593.736} C_VEL
LIN {X 0,Y 601.422,Z 240.378,A -85,B 0,C 180,E1 -596.064,E2 -596.064} C_VEL
LIN {X 0,Y 601.433,Z 240.374,A -85,B 0,C 180,E1 -598.541,E2 -598.541} C_VEL
LIN {X 0,Y 601.436,Z 240.381,A -85,B 0,C 180,E1 -601.374,E2 -601.374} C_VEL
LIN {X 0,Y 601.399,Z 240.388,A -85,B 0,C 180,E1 -603.636,E2 -603.636} C_VEL
LIN {X 0,Y 601.408,Z 240.377,A -85,B 0,C 180,E1 -606.59,E2 -606.59} C_VEL
LIN {X 0,Y 601.429,Z 240.384,A -85,B 0,C 180,E1 -609.478,E2 -609.478} C_VEL
LIN {X 0,Y 601.385,Z 240.381,A -85,B 0,C 180,E1 -612.311,E2 -612.311} C_VEL
LIN {X 0,Y 601.404,Z 240.378,A -85,B 0,C 180,E1 -614.409,E2 -614.409} C_VEL
LIN {X 0,Y 601.418,Z 240.38,A -85,B 0,C 180,E1 -617.172,E2 -617.172} C_VEL
LIN {X 0,Y 601.416,Z 240.381,A -85,B 0,C 180,E1 -619.905,E2 -619.905} C_VEL
LIN {X 0,Y 601.431,Z 240.374,A -85,B 0,C 180,E1 -622.615,E2 -622.615} C_VEL
LIN {X 0,Y 601.424,Z 240.381,A -85,B 0,C 180,E1 -625.308,E2 -625.308} C_VEL
LIN {X 0,Y 601.403,Z 240.382,A -85,B 0,C 180,E1 -627.991,E2 -627.991} C_VEL
LIN {X 0,Y 601.431,Z 240.374,A -85,B 0,C 180,E1 -630.669,E2 -630.669} C_VEL
LIN {X 0,Y 601.433,Z 240.381,A -85,B 0,C 180,E1 -633.349,E2 -633.349} C_VEL
LIN {X 0,Y 601.39,Z 240.383,A -85,B 0,C 180,E1 -636.037,E2 -636.037} C_VEL
LIN {X 0,Y 601.422,Z 240.378,A -85,B 0,C 180,E1 -638.061,E2 -638.061} C_VEL
LIN {X 0,Y 601.412,Z 240.379,A -85,B 0,C 180,E1 -641.011,E2 -641.011} C_VEL
LIN {X 0,Y 601.41,Z 240.387,A -85,B 0,C 180,E1 -643.516,E2 -643.516} C_VEL
LIN {X 0,Y 601.412,Z 240.378,A -85,B 0,C 180,E1 -646.287,E2 -646.287} C_VEL
LIN {X 0,Y 601.406,Z 240.38,A -85,B 0,C 180,E1 -649.099,E2 -649.099} C_VEL
LIN {X 0,Y 601.389,Z 240.384,A -85,B 0,C 180,E1 -651.959,E2 -651.959} C_VEL
LIN {X 0,Y 601.391,Z 240.38,A -85,B 0,C 180,E1 -654.286,E2 -654.286} C_VEL
LIN {X 0,Y 601.446,Z 240.375,A -85,B 0,C 180,E1 -657.111,E2 -657.111} C_VEL
LIN {X 0,Y 601.407,Z 240.385,A -85,B 0,C 180,E1 -659.393,E2 -659.393} C_VEL
LIN {X 0,Y 601.394,Z 240.388,A -85,B 0,C 180,E1 -661.726,E2 -661.726} C_VEL
LIN {X 0,Y 601.424,Z 240.438,A -85,B 0,C 180,E1 -663.147,E2 -663.147} C_VEL
LIN {X 0,Y 601.323,Z 253.095,A -85,B 0,C 180,E1 -666.004,E2 -666.004} C_VEL
LIN {X 0,Y 601.344,Z 265.185,A -85,B 0,C 180,E1 -668.706,E2 -668.706} C_VEL
LIN {X 0,Y 601.483,Z 318.398,A -85,B 0,C 180,E1 -669.348,E2 -669.348} C_VEL
LIN {X 0,Y 601.448,Z 341.407,A -85,B 0,C 180,E1 -669.645,E2 -669.645} C_VEL
LIN {X 0,Y 601.418,Z 353.124,A -85,B 0,C 180,E1 -669.922,E2 -669.922} C_VEL
LIN {X 0,Y 601.414,Z 363.541,A -85,B 0,C 180,E1 -670.307,E2 -670.307} C_VEL
LIN {X 0,Y 601.438,Z 371.576,A -85,B 0,C 180,E1 -670.693,E2 -670.693} C_VEL
LIN {X 0,Y 601.419,Z 380.088,A -85,B 0,C 180,E1 -671.206,E2 -671.206} C_VEL
LIN {X 0,Y 601.393,Z 387.664,A -85,B 0,C 180,E1 -671.767,E2 -671.767} C_VEL
LIN {X 0,Y 601.373,Z 394.744,A -85,B 0,C 180,E1 -672.403,E2 -672.403} C_VEL
LIN {X 0,Y 601.374,Z 401.299,A -85,B 0,C 180,E1 -673.119,E2 -673.119} C_VEL
LIN {X 0,Y 601.361,Z 408.221,A -85,B 0,C 180,E1 -674.055,E2 -674.055} C_VEL
LIN {X 0,Y 601.366,Z 413.552,A -85,B 0,C 180,E1 -675.007,E2 -675.007} C_VEL
LIN {X 0,Y 601.362,Z 417.495,A -85,B 0,C 180,E1 -675.945,E2 -675.945} C_VEL
LIN {X 0,Y 601.331,Z 420.31,A -85,B 0,C 180,E1 -676.881,E2 -676.881} C_VEL
LIN {X 0,Y 601.335,Z 421.52,A -85,B 0,C 180,E1 -677.416,E2 -677.416} C_VEL
LIN {X 0,Y 601.32,Z 422.733,A -85,B 0,C 180,E1 -678.417,E2 -678.417} C_VEL
LIN {X 0,Y 601.308,Z 422.842,A -85,B 0,C 180,E1 -679.437,E2 -679.437} C_VEL
LIN {X 0,Y 601.321,Z 421.805,A -85,B 0,C 180,E1 -680.476,E2 -680.476} C_VEL
LIN {X 0,Y 601.319,Z 419.506,A -85,B 0,C 180,E1 -681.541,E2 -681.541} C_VEL
LIN {X 0,Y 601.353,Z 415.616,A -85,B 0,C 180,E1 -682.626,E2 -682.626} C_VEL
LIN {X 0,Y 601.358,Z 411.824,A -85,B 0,C 180,E1 -683.415,E2 -683.415} C_VEL
LIN {X 0,Y 601.353,Z 406.767,A -85,B 0,C 180,E1 -684.244,E2 -684.244} C_VEL
LIN {X 0,Y 601.377,Z 400.492,A -85,B 0,C 180,E1 -685.067,E2 -685.067} C_VEL
LIN {X 0,Y 601.407,Z 392.78,A -85,B 0,C 180,E1 -685.881,E2 -685.881} C_VEL
LIN {X 0,Y 601.407,Z 384.386,A -85,B 0,C 180,E1 -686.586,E2 -686.586} C_VEL
LIN {X 0,Y 601.464,Z 375.112,A -85,B 0,C 180,E1 -687.196,E2 -687.196} C_VEL
LIN {X 0,Y 601.442,Z 366.776,A -85,B 0,C 180,E1 -687.635,E2 -687.635} C_VEL
LIN {X 0,Y 601.444,Z 358.469,A -85,B 0,C 180,E1 -687.981,E2 -687.981} C_VEL
LIN {X 0,Y 601.427,Z 349.022,A -85,B 0,C 180,E1 -688.276,E2 -688.276} C_VEL
LIN {X 0,Y 601.478,Z 339.364,A -85,B 0,C 180,E1 -688.478,E2 -688.478} C_VEL
LIN {X 0,Y 601.4,Z 265.296,A -85,B 0,C 180,E1 -689.374,E2 -689.374} C_VEL
LIN {X 0,Y 601.379,Z 252.886,A -85,B 0,C 180,E1 -692.131,E2 -692.131} C_VEL
LIN {X 0,Y 601.411,Z 240.38,A -85,B 0,C 180,E1 -694.984,E2 -694.984} C_VEL
LIN {X 0,Y 601.404,Z 240.378,A -85,B 0,C 180,E1 -697.394,E2 -697.394} C_VEL
LIN {X 0,Y 601.4,Z 240.384,A -85,B 0,C 180,E1 -700.191,E2 -700.191} C_VEL
LIN {X 0,Y 601.427,Z 240.378,A -85,B 0,C 180,E1 -703.015,E2 -703.015} C_VEL
LIN {X 0,Y 601.41,Z 240.379,A -85,B 0,C 180,E1 -705.908,E2 -705.908} C_VEL
LIN {X 0,Y 601.426,Z 240.385,A -85,B 0,C 180,E1 -708.542,E2 -708.542} C_VEL
LIN {X 0,Y 601.435,Z 240.375,A -85,B 0,C 180,E1 -711.263,E2 -711.263} C_VEL
LIN {X 0,Y 601.405,Z 240.38,A -85,B 0,C 180,E1 -713.963,E2 -713.963} C_VEL
LIN {X 0,Y 601.426,Z 240.383,A -85,B 0,C 180,E1 -716.651,E2 -716.651} C_VEL
LIN {X 0,Y 601.446,Z 240.373,A -85,B 0,C 180,E1 -719.331,E2 -719.331} C_VEL
LIN {X 0,Y 601.418,Z 240.379,A -85,B 0,C 180,E1 -722.01,E2 -722.01} C_VEL
LIN {X 0,Y 601.426,Z 240.382,A -85,B 0,C 180,E1 -724.692,E2 -724.692} C_VEL
LIN {X 0,Y 601.444,Z 240.373,A -85,B 0,C 180,E1 -727.386,E2 -727.386} C_VEL
LIN {X 0,Y 601.429,Z 240.379,A -85,B 0,C 180,E1 -730.096,E2 -730.096} C_VEL
LIN {X 0,Y 601.416,Z 240.381,A -85,B 0,C 180,E1 -732.829,E2 -732.829} C_VEL
LIN {X 0,Y 601.407,Z 240.377,A -85,B 0,C 180,E1 -735.592,E2 -735.592} C_VEL
LIN {X 0,Y 601.419,Z 240.385,A -85,B 0,C 180,E1 -738.392,E2 -738.392} C_VEL
LIN {X 0,Y 601.402,Z 240.378,A -85,B 0,C 180,E1 -741.24,E2 -741.24} C_VEL
LIN {X 0,Y 601.454,Z 240.376,A -85,B 0,C 180,E1 -744.141,E2 -744.141} C_VEL
LIN {X 0,Y 601.438,Z 240.375,A -85,B 0,C 180,E1 -747.112,E2 -747.112} C_VEL
LIN {X 0,Y 601.418,Z 240.376,A -85,B 0,C 180,E1 -749.393,E2 -749.393} C_VEL
LIN {X 0,Y 601.404,Z 240.378,A -85,B 0,C 180,E1 -751.727,E2 -751.727} C_VEL
LIN {X 0,Y 601.425,Z 240.379,A -85,B 0,C 180,E1 -754.119,E2 -754.119} C_VEL
LIN {X 0,Y 601.402,Z 240.387,A -85,B 0,C 180,E1 -756.583,E2 -756.583} C_VEL
LIN {X 0,Y 601.436,Z 240.374,A -85,B 0,C 180,E1 -759.537,E2 -759.537} C_VEL
LIN {X 0,Y 601.406,Z 240.386,A -85,B 0,C 180,E1 -762.592,E2 -762.592} C_VEL
LIN {X 0,Y 601.421,Z 240.376,A -85,B 0,C 180,E1 -765.483,E2 -765.483} C_VEL
LIN {X 0,Y 601.422,Z 240.385,A -85,B 0,C 180,E1 -768.407,E2 -768.407} C_VEL
LIN {X 0,Y 601.427,Z 240.375,A -85,B 0,C 180,E1 -771.53,E2 -771.53} C_VEL
LIN {X 0,Y 601.403,Z 240.384,A -85,B 0,C 180,E1 -774.247,E2 -774.247} C_VEL
LIN {X 0,Y 601.427,Z 240.382,A -85,B 0,C 180,E1 -776.687,E2 -776.687} C_VEL
LIN {X 0,Y 601.407,Z 240.379,A -85,B 0,C 180,E1 -779.058,E2 -779.058} C_VEL
LIN {X 0,Y 601.414,Z 240.377,A -85,B 0,C 180,E1 -781.373,E2 -781.373} C_VEL
LIN {X 0,Y 601.414,Z 240.381,A -85,B 0,C 180,E1 -784.133,E2 -784.133} C_VEL
LIN {X 0,Y 601.413,Z 240.387,A -85,B 0,C 180,E1 -786.59,E2 -786.59} C_VEL
LIN {X 0,Y 601.412,Z 240.489,A -85,B 0,C 180,E1 -787.58,E2 -787.58} C_VEL
LIN {X 0,Y 601.607,Z 245.894,A -85,B 0,C 180,E1 -788.409,E2 -788.409} C_VEL
LIN {X 0,Y 601.505,Z 262.509,A -85,B 0,C 180,E1 -790.905,E2 -790.905} C_VEL
LIN {X 0,Y 601.515,Z 281.498,A -85,B 0,C 180,E1 -793.716,E2 -793.716} C_VEL
LIN {X 0,Y 601.43,Z 301.675,A -85,B 0,C 180,E1 -796.657,E2 -796.657} C_VEL
LIN {X 0,Y 601.372,Z 319.477,A -85,B 0,C 180,E1 -799.223,E2 -799.223} C_VEL
LIN {X 0,Y 601.389,Z 322.296,A -85,B 0,C 180,E1 -799.628,E2 -799.628} C_VEL
LIN {X 0,Y 601.469,Z 400.464,A -85,B 0,C 180,E1 -800.585,E2 -800.585} C_VEL
LIN {X 0,Y 601.432,Z 410.918,A -85,B 0,C 180,E1 -800.818,E2 -800.818} C_VEL
LIN {X 0,Y 601.414,Z 423.544,A -85,B 0,C 180,E1 -801.262,E2 -801.262} C_VEL
LIN {X 0,Y 601.437,Z 432.241,A -85,B 0,C 180,E1 -801.686,E2 -801.686} C_VEL
LIN {X 0,Y 601.402,Z 440.548,A -85,B 0,C 180,E1 -802.193,E2 -802.193} C_VEL
LIN {X 0,Y 601.409,Z 448.405,A -85,B 0,C 180,E1 -802.784,E2 -802.784} C_VEL
LIN {X 0,Y 601.412,Z 455.599,A -85,B 0,C 180,E1 -803.443,E2 -803.443} C_VEL
LIN {X 0,Y 601.391,Z 463.193,A -85,B 0,C 180,E1 -804.3,E2 -804.3} C_VEL
LIN {X 0,Y 601.38,Z 469.029,A -85,B 0,C 180,E1 -805.14,E2 -805.14} C_VEL
LIN {X 0,Y 601.345,Z 473.632,A -85,B 0,C 180,E1 -805.979,E2 -805.979} C_VEL
LIN {X 0,Y 601.344,Z 476.622,A -85,B 0,C 180,E1 -806.65,E2 -806.65} C_VEL
LIN {X 0,Y 601.326,Z 478.932,A -85,B 0,C 180,E1 -807.321,E2 -807.321} C_VEL
LIN {X 0,Y 601.343,Z 480.679,A -85,B 0,C 180,E1 -807.991,E2 -807.991} C_VEL
LIN {X 0,Y 601.345,Z 481.935,A -85,B 0,C 180,E1 -808.661,E2 -808.661} C_VEL
LIN {X 0,Y 601.335,Z 482.713,A -85,B 0,C 180,E1 -809.331,E2 -809.331} C_VEL
LIN {X 0,Y 601.332,Z 483,A -85,B 0,C 180,E1 -810,E2 -810} C_VEL
LIN {X 0,Y 601.335,Z 482.713,A -85,B 0,C 180,E1 -810.67,E2 -810.67} C_VEL
LIN {X 0,Y 601.345,Z 481.934,A -85,B 0,C 180,E1 -811.34,E2 -811.34} C_VEL
LIN {X 0,Y 601.343,Z 480.678,A -85,B 0,C 180,E1 -812.009,E2 -812.009} C_VEL
LIN {X 0,Y 601.343,Z 477.786,A -85,B 0,C 180,E1 -813.015,E2 -813.015} C_VEL
LIN {X 0,Y 601.365,Z 475.146,A -85,B 0,C 180,E1 -813.685,E2 -813.685} C_VEL
LIN {X 0,Y 601.341,Z 469.984,A -85,B 0,C 180,E1 -814.693,E2 -814.693} C_VEL
LIN {X 0,Y 601.383,Z 464.429,A -85,B 0,C 180,E1 -815.533,E2 -815.533} C_VEL
LIN {X 0,Y 601.394,Z 457.153,A -85,B 0,C 180,E1 -816.403,E2 -816.403} C_VEL
LIN {X 0,Y 601.413,Z 449.416,A -85,B 0,C 180,E1 -817.132,E2 -817.132} C_VEL
LIN {X 0,Y 601.424,Z 441.762,A -85,B 0,C 180,E1 -817.723,E2 -817.723} C_VEL
LIN {X 0,Y 601.445,Z 433.722,A -85,B 0,C 180,E1 -818.23,E2 -818.23} C_VEL
LIN {X 0,Y 601.428,Z 425.392,A -85,B 0,C 180,E1 -818.653,E2 -818.653} C_VEL
LIN {X 0,Y 601.423,Z 416.89,A -85,B 0,C 180,E1 -818.992,E2 -818.992} C_VEL
LIN {X 0,Y 601.451,Z 406.755,A -85,B 0,C 180,E1 -819.288,E2 -819.288} C_VEL
LIN {X 0,Y 601.485,Z 395.06,A -85,B 0,C 180,E1 -819.5,E2 -819.5} C_VEL
LIN {X 0,Y 601.389,Z 322.293,A -85,B 0,C 180,E1 -820.372,E2 -820.372} C_VEL
LIN {X 0,Y 601.46,Z 302.859,A -85,B 0,C 180,E1 -823.171,E2 -823.171} C_VEL
LIN {X 0,Y 601.475,Z 282.683,A -85,B 0,C 180,E1 -826.111,E2 -826.111} C_VEL
LIN {X 0,Y 601.507,Z 264.197,A -85,B 0,C 180,E1 -828.844,E2 -828.844} C_VEL
LIN {X 0,Y 601.589,Z 247.078,A -85,B 0,C 180,E1 -831.412,E2 -831.412} C_VEL
LIN {X 0,Y 601.557,Z 241.191,A -85,B 0,C 180,E1 -832.307,E2 -832.307} C_VEL
LIN {X 0,Y 601.436,Z 240.378,A -85,B 0,C 180,E1 -832.473,E2 -832.473} C_VEL
LIN {X 0,Y 601.394,Z 240.381,A -85,B 0,C 180,E1 -834.879,E2 -834.879} C_VEL
LIN {X 0,Y 601.406,Z 240.386,A -85,B 0,C 180,E1 -837.361,E2 -837.361} C_VEL
LIN {X 0,Y 601.428,Z 240.376,A -85,B 0,C 180,E1 -840.164,E2 -840.164} C_VEL
LIN {X 0,Y 601.412,Z 240.377,A -85,B 0,C 180,E1 -842.714,E2 -842.714} C_VEL
LIN {X 0,Y 601.385,Z 240.384,A -85,B 0,C 180,E1 -845.11,E2 -845.11} C_VEL
LIN {X 0,Y 601.431,Z 240.383,A -85,B 0,C 180,E1 -847.419,E2 -847.419} C_VEL
LIN {X 0,Y 601.399,Z 240.381,A -85,B 0,C 180,E1 -849.995,E2 -849.995} C_VEL
LIN {X 0,Y 601.405,Z 240.378,A -85,B 0,C 180,E1 -852.67,E2 -852.67} C_VEL
LIN {X 0,Y 601.423,Z 240.386,A -85,B 0,C 180,E1 -855.482,E2 -855.482} C_VEL
LIN {X 0,Y 601.416,Z 240.376,A -85,B 0,C 180,E1 -858.407,E2 -858.407} C_VEL
LIN {X 0,Y 601.405,Z 240.379,A -85,B 0,C 180,E1 -860.873,E2 -860.873} C_VEL
LIN {X 0,Y 601.439,Z 240.38,A -85,B 0,C 180,E1 -863.733,E2 -863.733} C_VEL
LIN {X 0,Y 601.422,Z 240.376,A -85,B 0,C 180,E1 -866.686,E2 -866.686} C_VEL
LIN {X 0,Y 601.406,Z 240.38,A -85,B 0,C 180,E1 -869.057,E2 -869.057} C_VEL
LIN {X 0,Y 601.43,Z 240.382,A -85,B 0,C 180,E1 -871.373,E2 -871.373} C_VEL
LIN {X 0,Y 601.418,Z 240.378,A -85,B 0,C 180,E1 -874.13,E2 -874.13} C_VEL
LIN {X 0,Y 601.415,Z 240.376,A -85,B 0,C 180,E1 -876.589,E2 -876.589} C_VEL
LIN {X 0,Y 601.43,Z 240.384,A -85,B 0,C 180,E1 -879.478,E2 -879.478} C_VEL
LIN {X 0,Y 601.391,Z 240.38,A -85,B 0,C 180,E1 -882.311,E2 -882.311} C_VEL
LIN {X 0,Y 601.408,Z 240.377,A -85,B 0,C 180,E1 -884.408,E2 -884.408} C_VEL
LIN {X 0,Y 601.415,Z 240.381,A -85,B 0,C 180,E1 -887.171,E2 -887.171} C_VEL
LIN {X 0,Y 601.431,Z 240.379,A -85,B 0,C 180,E1 -889.904,E2 -889.904} C_VEL
LIN {X 0,Y 601.434,Z 240.374,A -85,B 0,C 180,E1 -892.614,E2 -892.614} C_VEL
LIN {X 0,Y 601.424,Z 240.382,A -85,B 0,C 180,E1 -895.307,E2 -895.307} C_VEL
LIN {X 0,Y 601.42,Z 240.379,A -85,B 0,C 180,E1 -897.99,E2 -897.99} C_VEL
LIN {X 0,Y 601.449,Z 240.372,A -85,B 0,C 180,E1 -900.669,E2 -900.669} C_VEL
LIN {X 0,Y 601.425,Z 240.382,A -85,B 0,C 180,E1 -903.349,E2 -903.349} C_VEL
LIN {X 0,Y 601.407,Z 240.38,A -85,B 0,C 180,E1 -906.037,E2 -906.037} C_VEL
LIN {X 0,Y 601.435,Z 240.374,A -85,B 0,C 180,E1 -908.737,E2 -908.737} C_VEL
LIN {X 0,Y 601.427,Z 240.384,A -85,B 0,C 180,E1 -911.458,E2 -911.458} C_VEL
LIN {X 0,Y 601.406,Z 240.378,A -85,B 0,C 180,E1 -912.385,E2 -912.385} C_VEL
LIN {X 0,Y 600.743,Z 240.462,A -85,B 0,C 180,E1 -912.945,E2 -912.945} C_VEL
LIN {X 0,Y 597.892,Z 240.821,A -85,B 0,C 180,E1 -913.852,E2 -913.852} C_VEL
LIN {X 0,Y 595.48,Z 241.12,A -85,B 0,C 180,E1 -914.582,E2 -914.582} C_VEL
LIN {X 0,Y 594.442,Z 241.249,A -85,B 0,C 180,E1 -915.146,E2 -915.146} C_VEL
LIN {X 0,Y 594.356,Z 241.259,A -85,B 0,C 180,E1 -915.337,E2 -915.337} C_VEL
LIN {X 0,Y 594.373,Z 241.258,A -85,B 0,C 180,E1 -917.904,E2 -917.904} C_VEL
LIN {X 0,Y 594.377,Z 241.255,A -85,B 0,C 180,E1 -920.918,E2 -920.918} C_VEL
LIN {X 0,Y 594.382,Z 241.261,A -85,B 0,C 180,E1 -923.703,E2 -923.703} C_VEL
LIN {X 0,Y 594.378,Z 241.253,A -85,B 0,C 180,E1 -926.699,E2 -926.699} C_VEL
LIN {X 0,Y 594.377,Z 241.255,A -85,B 0,C 180,E1 -928.998,E2 -928.998} C_VEL
LIN {X 0,Y 594.384,Z 241.261,A -85,B 0,C 180,E1 -931.645,E2 -931.645} C_VEL
LIN {X 0,Y 594.392,Z 241.251,A -85,B 0,C 180,E1 -934.578,E2 -934.578} C_VEL
LIN {X 0,Y 594.377,Z 241.256,A -85,B 0,C 180,E1 -937.086,E2 -937.086} C_VEL
LIN {X 0,Y 594.367,Z 241.261,A -85,B 0,C 180,E1 -939.774,E2 -939.774} C_VEL
LIN {X 0,Y 594.359,Z 241.256,A -85,B 0,C 180,E1 -942.375,E2 -942.375} C_VEL
LIN {X 0,Y 594.352,Z 241.261,A -85,B 0,C 180,E1 -945.191,E2 -945.191} C_VEL
LIN {X 0,Y 594.379,Z 241.263,A -85,B 0,C 180,E1 -947.626,E2 -947.626} C_VEL
LIN {X 0,Y 594.382,Z 241.253,A -85,B 0,C 180,E1 -950.321,E2 -950.321} C_VEL
LIN {X 0,Y 594.376,Z 241.255,A -85,B 0,C 180,E1 -952.913,E2 -952.913} C_VEL
LIN {X 0,Y 594.375,Z 241.259,A -85,B 0,C 180,E1 -955.861,E2 -955.861} C_VEL
LIN {X 0,Y 594.382,Z 241.253,A -85,B 0,C 180,E1 -958.651,E2 -958.651} C_VEL
LIN {X 0,Y 594.378,Z 241.255,A -85,B 0,C 180,E1 -961.041,E2 -961.041} C_VEL
LIN {X 0,Y 594.373,Z 241.257,A -85,B 0,C 180,E1 -963.977,E2 -963.977} C_VEL
LIN {X 0,Y 594.378,Z 241.254,A -85,B 0,C 180,E1 -966.296,E2 -966.296} C_VEL
LIN {X 0,Y 594.403,Z 241.255,A -85,B 0,C 180,E1 -969.225,E2 -969.225} C_VEL
LIN {X 0,Y 594.343,Z 241.26,A -85,B 0,C 180,E1 -972.095,E2 -972.095} C_VEL
LIN {X 0,Y 594.358,Z 241.257,A -85,B 0,C 180,E1 -974.219,E2 -974.219} C_VEL
LIN {X 0,Y 594.363,Z 241.257,A -85,B 0,C 180,E1 -977.017,E2 -977.017} C_VEL
LIN {X 0,Y 594.38,Z 241.26,A -85,B 0,C 180,E1 -979.784,E2 -979.784} C_VEL
LIN {X 0,Y 594.383,Z 241.252,A -85,B 0,C 180,E1 -982.527,E2 -982.527} C_VEL
LIN {X 0,Y 594.391,Z 241.256,A -85,B 0,C 180,E1 -985.252,E2 -985.252} C_VEL
LIN {X 0,Y 594.375,Z 241.258,A -85,B 0,C 180,E1 -987.967,E2 -987.967} C_VEL
LIN {X 0,Y 594.403,Z 241.25,A -85,B 0,C 180,E1 -990.677,E2 -990.677} C_VEL
LIN {X 0,Y 594.382,Z 241.26,A -85,B 0,C 180,E1 -993.389,E2 -993.389} C_VEL
LIN {X 0,Y 594.341,Z 241.26,A -85,B 0,C 180,E1 -996.109,E2 -996.109} C_VEL
LIN {X 0,Y 594.368,Z 241.256,A -85,B 0,C 180,E1 -998.157,E2 -998.157} C_VEL
LIN {X 0,Y 594.376,Z 241.256,A -85,B 0,C 180,E1 -1001.072,E2 -1001.072} C_VEL
LIN {X 0,Y 594.368,Z 241.263,A -85,B 0,C 180,E1 -1003.679,E2 -1003.679} C_VEL
LIN {X 0,Y 594.372,Z 241.254,A -85,B 0,C 180,E1 -1006.486,E2 -1006.486} C_VEL
LIN {X 0,Y 594.356,Z 241.262,A -85,B 0,C 180,E1 -1009.334,E2 -1009.334} C_VEL
LIN {X 0,Y 594.351,Z 241.266,A -85,B 0,C 180,E1 -1011.503,E2 -1011.503} C_VEL
LIN {X 0,Y 594.354,Z 241.256,A -85,B 0,C 180,E1 -1014.447,E2 -1014.447} C_VEL
LIN {X 0,Y 594.372,Z 241.254,A -85,B 0,C 180,E1 -1016.699,E2 -1016.699} C_VEL
LIN {X 0,Y 594.366,Z 241.256,A -85,B 0,C 180,E1 -1018.998,E2 -1018.998} C_VEL
LIN {X 0,Y 594.376,Z 241.264,A -85,B 0,C 180,E1 -1021.644,E2 -1021.644} C_VEL
LIN {X 0,Y 594.366,Z 241.303,A -85,B 0,C 180,E1 -1023.152,E2 -1023.152} C_VEL
LIN {X 0,Y 594.277,Z 253.02,A -85,B 0,C 180,E1 -1025.83,E2 -1025.83} C_VEL
LIN {X 0,Y 594.267,Z 264.79,A -85,B 0,C 180,E1 -1028.493,E2 -1028.493} C_VEL
LIN {X 0,Y 594.261,Z 265.201,A -85,B 0,C 180,E1 -1028.585,E2 -1028.585} C_VEL
LIN {X 0,Y 594.544,Z 271.627,A -85,B 0,C 180,E1 -1028.671,E2 -1028.671} C_VEL
LIN {X 0,Y 594.449,Z 339.891,A -85,B 0,C 180,E1 -1029.509,E2 -1029.509} C_VEL
LIN {X 0,Y 594.421,Z 349.5,A -85,B 0,C 180,E1 -1029.717,E2 -1029.717} C_VEL
LIN {X 0,Y 594.395,Z 359.366,A -85,B 0,C 180,E1 -1030.034,E2 -1030.034} C_VEL
LIN {X 0,Y 594.39,Z 371.059,A -85,B 0,C 180,E1 -1030.564,E2 -1030.564} C_VEL
LIN {X 0,Y 594.373,Z 380.148,A -85,B 0,C 180,E1 -1031.116,E2 -1031.116} C_VEL
LIN {X 0,Y 594.364,Z 387.37,A -85,B 0,C 180,E1 -1031.655,E2 -1031.655} C_VEL
LIN {X 0,Y 594.311,Z 395.296,A -85,B 0,C 180,E1 -1032.379,E2 -1032.379} C_VEL
LIN {X 0,Y 594.293,Z 402.388,A -85,B 0,C 180,E1 -1033.179,E2 -1033.179} C_VEL
LIN {X 0,Y 594.293,Z 409.685,A -85,B 0,C 180,E1 -1034.243,E2 -1034.243} C_VEL
LIN {X 0,Y 594.288,Z 412.817,A -85,B 0,C 180,E1 -1034.803,E2 -1034.803} C_VEL
LIN {X 0,Y 594.256,Z 416.972,A -85,B 0,C 180,E1 -1035.753,E2 -1035.753} C_VEL
LIN {X 0,Y 594.243,Z 419.921,A -85,B 0,C 180,E1 -1036.691,E2 -1036.691} C_VEL
LIN {X 0,Y 594.245,Z 421.832,A -85,B 0,C 180,E1 -1037.615,E2 -1037.615} C_VEL
LIN {X 0,Y 594.213,Z 422.785,A -85,B 0,C 180,E1 -1038.523,E2 -1038.523} C_VEL
LIN {X 0,Y 594.23,Z 422.851,A -85,B 0,C 180,E1 -1039.423,E2 -1039.423} C_VEL
LIN {X 0,Y 594.222,Z 422.063,A -85,B 0,C 180,E1 -1040.308,E2 -1040.308} C_VEL
LIN {X 0,Y 594.234,Z 420.129,A -85,B 0,C 180,E1 -1041.312,E2 -1041.312} C_VEL
LIN {X 0,Y 594.247,Z 416.724,A -85,B 0,C 180,E1 -1042.408,E2 -1042.408} C_VEL
LIN {X 0,Y 594.296,Z 413.029,A -85,B 0,C 180,E1 -1043.245,E2 -1043.245} C_VEL
LIN {X 0,Y 594.284,Z 407.701,A -85,B 0,C 180,E1 -1044.171,E2 -1044.171} C_VEL
LIN {X 0,Y 594.299,Z 401.622,A -85,B 0,C 180,E1 -1045.003,E2 -1045.003} C_VEL
LIN {X 0,Y 594.329,Z 395.712,A -85,B 0,C 180,E1 -1045.669,E2 -1045.669} C_VEL
LIN {X 0,Y 594.349,Z 388.499,A -85,B 0,C 180,E1 -1046.34,E2 -1046.34} C_VEL
LIN {X 0,Y 594.398,Z 380.463,A -85,B 0,C 180,E1 -1046.951,E2 -1046.951} C_VEL
LIN {X 0,Y 594.447,Z 370.474,A -85,B 0,C 180,E1 -1047.558,E2 -1047.558} C_VEL
LIN {X 0,Y 594.435,Z 359.06,A -85,B 0,C 180,E1 -1048.066,E2 -1048.066} C_VEL
LIN {X 0,Y 594.444,Z 349.754,A -85,B 0,C 180,E1 -1048.366,E2 -1048.366} C_VEL
LIN {X 0,Y 594.467,Z 340.578,A -85,B 0,C 180,E1 -1048.57,E2 -1048.57} C_VEL
LIN {X 0,Y 594.558,Z 288.325,A -85,B 0,C 180,E1 -1049.218,E2 -1049.218} C_VEL
LIN {X 0,Y 594.42,Z 266.216,A -85,B 0,C 180,E1 -1049.486,E2 -1049.486} C_VEL
LIN {X 0,Y 594.296,Z 265.125,A -85,B 0,C 180,E1 -1049.521,E2 -1049.521} C_VEL
LIN {X 0,Y 594.308,Z 253.482,A -85,B 0,C 180,E1 -1052.155,E2 -1052.155} C_VEL
LIN {X 0,Y 594.372,Z 241.257,A -85,B 0,C 180,E1 -1054.971,E2 -1054.971} C_VEL
LIN {X 0,Y 594.353,Z 241.257,A -85,B 0,C 180,E1 -1057.767,E2 -1057.767} C_VEL
LIN {X 0,Y 594.369,Z 241.257,A -85,B 0,C 180,E1 -1059.947,E2 -1059.947} C_VEL
LIN {X 0,Y 594.383,Z 241.258,A -85,B 0,C 180,E1 -1062.807,E2 -1062.807} C_VEL
LIN {X 0,Y 594.377,Z 241.254,A -85,B 0,C 180,E1 -1065.826,E2 -1065.826} C_VEL
LIN {X 0,Y 594.385,Z 241.261,A -85,B 0,C 180,E1 -1068.405,E2 -1068.405} C_VEL
LIN {X 0,Y 594.395,Z 241.252,A -85,B 0,C 180,E1 -1071.159,E2 -1071.159} C_VEL
LIN {X 0,Y 594.361,Z 241.257,A -85,B 0,C 180,E1 -1073.892,E2 -1073.892} C_VEL
LIN {X 0,Y 594.378,Z 241.262,A -85,B 0,C 180,E1 -1076.611,E2 -1076.611} C_VEL
LIN {X 0,Y 594.416,Z 241.249,A -85,B 0,C 180,E1 -1079.323,E2 -1079.323} C_VEL
LIN {X 0,Y 594.388,Z 241.255,A -85,B 0,C 180,E1 -1082.033,E2 -1082.033} C_VEL
LIN {X 0,Y 594.394,Z 241.257,A -85,B 0,C 180,E1 -1084.748,E2 -1084.748} C_VEL
LIN {X 0,Y 594.393,Z 241.251,A -85,B 0,C 180,E1 -1087.474,E2 -1087.474} C_VEL
LIN {X 0,Y 594.388,Z 241.257,A -85,B 0,C 180,E1 -1090.216,E2 -1090.216} C_VEL
LIN {X 0,Y 594.362,Z 241.258,A -85,B 0,C 180,E1 -1092.984,E2 -1092.984} C_VEL
LIN {X 0,Y 594.362,Z 241.256,A -85,B 0,C 180,E1 -1095.781,E2 -1095.781} C_VEL
LIN {X 0,Y 594.382,Z 241.261,A -85,B 0,C 180,E1 -1098.618,E2 -1098.618} C_VEL
LIN {X 0,Y 594.361,Z 241.255,A -85,B 0,C 180,E1 -1101.504,E2 -1101.504} C_VEL
LIN {X 0,Y 594.381,Z 241.263,A -85,B 0,C 180,E1 -1104.447,E2 -1104.447} C_VEL
LIN {X 0,Y 594.378,Z 241.26,A -85,B 0,C 180,E1 -1106.7,E2 -1106.7} C_VEL
LIN {X 0,Y 594.377,Z 241.255,A -85,B 0,C 180,E1 -1108.999,E2 -1108.999} C_VEL
LIN {X 0,Y 594.379,Z 241.253,A -85,B 0,C 180,E1 -1111.645,E2 -1111.645} C_VEL
LIN {X 0,Y 594.386,Z 241.261,A -85,B 0,C 180,E1 -1114.58,E2 -1114.58} C_VEL
LIN {X 0,Y 594.377,Z 241.255,A -85,B 0,C 180,E1 -1117.088,E2 -1117.088} C_VEL
LIN {X 0,Y 594.372,Z 241.255,A -85,B 0,C 180,E1 -1119.776,E2 -1119.776} C_VEL
LIN {X 0,Y 594.363,Z 241.264,A -85,B 0,C 180,E1 -1122.376,E2 -1122.376} C_VEL
LIN {X 0,Y 594.358,Z 241.256,A -85,B 0,C 180,E1 -1125.192,E2 -1125.192} C_VEL
LIN {X 0,Y 594.382,Z 241.257,A -85,B 0,C 180,E1 -1128.152,E2 -1128.152} C_VEL
LIN {X 0,Y 594.372,Z 241.255,A -85,B 0,C 180,E1 -1131.195,E2 -1131.195} C_VEL
LIN {X 0,Y 594.39,Z 241.252,A -85,B 0,C 180,E1 -1133.759,E2 -1133.759} C_VEL
LIN {X 0,Y 594.381,Z 241.259,A -85,B 0,C 180,E1 -1136.24,E2 -1136.24} C_VEL
LIN {X 0,Y 594.366,Z 241.263,A -85,B 0,C 180,E1 -1138.65,E2 -1138.65} C_VEL
LIN {X 0,Y 594.375,Z 241.256,A -85,B 0,C 180,E1 -1141.044,E2 -1141.044} C_VEL
LIN {X 0,Y 594.365,Z 241.258,A -85,B 0,C 180,E1 -1143.982,E2 -1143.982} C_VEL
LIN {X 0,Y 594.388,Z 241.26,A -85,B 0,C 180,E1 -1146.297,E2 -1146.297} C_VEL
LIN {X 0,Y 594.417,Z 241.429,A -85,B 0,C 180,E1 -1147.447,E2 -1147.447} C_VEL
LIN {X 0,Y 594.701,Z 245.894,A -85,B 0,C 180,E1 -1148.146,E2 -1148.146} C_VEL
LIN {X 0,Y 594.568,Z 262.509,A -85,B 0,C 180,E1 -1150.673,E2 -1150.673} C_VEL
LIN {X 0,Y 594.508,Z 281.498,A -85,B 0,C 180,E1 -1153.518,E2 -1153.518} C_VEL
LIN {X 0,Y 594.399,Z 300.488,A -85,B 0,C 180,E1 -1156.322,E2 -1156.322} C_VEL
LIN {X 0,Y 594.348,Z 317.341,A -85,B 0,C 180,E1 -1158.784,E2 -1158.784} C_VEL
LIN {X 0,Y 594.338,Z 322.296,A -85,B 0,C 180,E1 -1159.504,E2 -1159.504} C_VEL
LIN {X 0,Y 594.576,Z 332.485,A -85,B 0,C 180,E1 -1159.637,E2 -1159.637} C_VEL
LIN {X 0,Y 594.5,Z 399.163,A -85,B 0,C 180,E1 -1160.452,E2 -1160.452} C_VEL
LIN {X 0,Y 594.444,Z 408.428,A -85,B 0,C 180,E1 -1160.645,E2 -1160.645} C_VEL
LIN {X 0,Y 594.413,Z 416.9,A -85,B 0,C 180,E1 -1160.902,E2 -1160.902} C_VEL
LIN {X 0,Y 594.391,Z 425.403,A -85,B 0,C 180,E1 -1161.244,E2 -1161.244} C_VEL
LIN {X 0,Y 594.42,Z 433.731,A -85,B 0,C 180,E1 -1161.673,E2 -1161.673} C_VEL
LIN {X 0,Y 594.359,Z 441.768,A -85,B 0,C 180,E1 -1162.185,E2 -1162.185} C_VEL
LIN {X 0,Y 594.354,Z 449.419,A -85,B 0,C 180,E1 -1162.783,E2 -1162.783} C_VEL
LIN {X 0,Y 594.33,Z 457.811,A -85,B 0,C 180,E1 -1163.59,E2 -1163.59} C_VEL
LIN {X 0,Y 594.309,Z 464.433,A -85,B 0,C 180,E1 -1164.402,E2 -1164.402} C_VEL
LIN {X 0,Y 594.256,Z 469.988,A -85,B 0,C 180,E1 -1165.252,E2 -1165.252} C_VEL
LIN {X 0,Y 594.287,Z 475.148,A -85,B 0,C 180,E1 -1166.271,E2 -1166.271} C_VEL
LIN {X 0,Y 594.246,Z 477.788,A -85,B 0,C 180,E1 -1166.949,E2 -1166.949} C_VEL
LIN {X 0,Y 594.242,Z 480.68,A -85,B 0,C 180,E1 -1167.967,E2 -1167.967} C_VEL
LIN {X 0,Y 594.245,Z 481.935,A -85,B 0,C 180,E1 -1168.645,E2 -1168.645} C_VEL
LIN {X 0,Y 594.235,Z 482.713,A -85,B 0,C 180,E1 -1169.323,E2 -1169.323} C_VEL
LIN {X 0,Y 594.233,Z 483,A -85,B 0,C 180,E1 -1170,E2 -1170} C_VEL
LIN {X 0,Y 594.235,Z 482.712,A -85,B 0,C 180,E1 -1170.678,E2 -1170.678} C_VEL
LIN {X 0,Y 594.245,Z 481.935,A -85,B 0,C 180,E1 -1171.356,E2 -1171.356} C_VEL
LIN {X 0,Y 594.242,Z 480.679,A -85,B 0,C 180,E1 -1172.033,E2 -1172.033} C_VEL
LIN {X 0,Y 594.246,Z 477.787,A -85,B 0,C 180,E1 -1173.051,E2 -1173.051} C_VEL
LIN {X 0,Y 594.287,Z 475.146,A -85,B 0,C 180,E1 -1173.729,E2 -1173.729} C_VEL
LIN {X 0,Y 594.256,Z 469.985,A -85,B 0,C 180,E1 -1174.749,E2 -1174.749} C_VEL
LIN {X 0,Y 594.309,Z 464.43,A -85,B 0,C 180,E1 -1175.599,E2 -1175.599} C_VEL
LIN {X 0,Y 594.345,Z 457.152,A -85,B 0,C 180,E1 -1176.479,E2 -1176.479} C_VEL
LIN {X 0,Y 594.354,Z 449.417,A -85,B 0,C 180,E1 -1177.218,E2 -1177.218} C_VEL
LIN {X 0,Y 594.359,Z 441.765,A -85,B 0,C 180,E1 -1177.815,E2 -1177.815} C_VEL
LIN {X 0,Y 594.42,Z 433.725,A -85,B 0,C 180,E1 -1178.328,E2 -1178.328} C_VEL
LIN {X 0,Y 594.392,Z 425.396,A -85,B 0,C 180,E1 -1178.756,E2 -1178.756} C_VEL
LIN {X 0,Y 594.413,Z 416.892,A -85,B 0,C 180,E1 -1179.099,E2 -1179.099} C_VEL
LIN {X 0,Y 594.46,Z 406.755,A -85,B 0,C 180,E1 -1179.398,E2 -1179.398} C_VEL
LIN {X 0,Y 594.501,Z 395.06,A -85,B 0,C 180,E1 -1179.612,E2 -1179.612} C_VEL
LIN {X 0,Y 594.377,Z 322.62,A -85,B 0,C 180,E1 -1180.485,E2 -1180.485} C_VEL
LIN {X 0,Y 594.315,Z 319.475,A -85,B 0,C 180,E1 -1180.906,E2 -1180.906} C_VEL
LIN {X 0,Y 594.423,Z 302.859,A -85,B 0,C 180,E1 -1183.33,E2 -1183.33} C_VEL
LIN {X 0,Y 594.504,Z 282.683,A -85,B 0,C 180,E1 -1186.306,E2 -1186.306} C_VEL
LIN {X 0,Y 594.528,Z 264.059,A -85,B 0,C 180,E1 -1189.094,E2 -1189.094} C_VEL
LIN {X 0,Y 594.663,Z 248.265,A -85,B 0,C 180,E1 -1191.492,E2 -1191.492} C_VEL
LIN {X 0,Y 594.718,Z 243.518,A -85,B 0,C 180,E1 -1192.219,E2 -1192.219} C_VEL
LIN {X 0,Y 594.391,Z 241.257,A -85,B 0,C 180,E1 -1192.589,E2 -1192.589} C_VEL
LIN {X 0,Y 594.373,Z 241.259,A -85,B 0,C 180,E1 -1195.193,E2 -1195.193} C_VEL
LIN {X 0,Y 594.367,Z 241.265,A -85,B 0,C 180,E1 -1197.523,E2 -1197.523} C_VEL
LIN {X 0,Y 594.385,Z 241.252,A -85,B 0,C 180,E1 -1200.328,E2 -1200.328} C_VEL
LIN {X 0,Y 594.376,Z 241.255,A -85,B 0,C 180,E1 -1202.95,E2 -1202.95} C_VEL
LIN {X 0,Y 594.352,Z 241.265,A -85,B 0,C 180,E1 -1205.408,E2 -1205.408} C_VEL
LIN {X 0,Y 594.384,Z 241.256,A -85,B 0,C 180,E1 -1207.94,E2 -1207.94} C_VEL
LIN {X 0,Y 594.37,Z 241.255,A -85,B 0,C 180,E1 -1210.821,E2 -1210.821} C_VEL
LIN {X 0,Y 594.363,Z 241.261,A -85,B 0,C 180,E1 -1213.299,E2 -1213.299} C_VEL
LIN {X 0,Y 594.364,Z 241.256,A -85,B 0,C 180,E1 -1216.16,E2 -1216.16} C_VEL
LIN {X 0,Y 594.373,Z 241.253,A -85,B 0,C 180,E1 -1218.535,E2 -1218.535} C_VEL
LIN {X 0,Y 594.377,Z 241.26,A -85,B 0,C 180,E1 -1221.295,E2 -1221.295} C_VEL
LIN {X 0,Y 594.391,Z 241.258,A -85,B 0,C 180,E1 -1223.758,E2 -1223.758} C_VEL
LIN {X 0,Y 594.375,Z 241.254,A -85,B 0,C 180,E1 -1226.238,E2 -1226.238} C_VEL
LIN {X 0,Y 594.364,Z 241.255,A -85,B 0,C 180,E1 -1228.649,E2 -1228.649} C_VEL
LIN {X 0,Y 594.379,Z 241.256,A -85,B 0,C 180,E1 -1231.041,E2 -1231.041} C_VEL
LIN {X 0,Y 594.39,Z 241.255,A -85,B 0,C 180,E1 -1233.975,E2 -1233.975} C_VEL
LIN {X 0,Y 594.386,Z 241.252,A -85,B 0,C 180,E1 -1236.295,E2 -1236.295} C_VEL
LIN {X 0,Y 594.402,Z 241.255,A -85,B 0,C 180,E1 -1239.224,E2 -1239.224} C_VEL
LIN {X 0,Y 594.349,Z 241.259,A -85,B 0,C 180,E1 -1242.094,E2 -1242.094} C_VEL
LIN {X 0,Y 594.363,Z 241.256,A -85,B 0,C 180,E1 -1244.219,E2 -1244.219} C_VEL
LIN {X 0,Y 594.361,Z 241.258,A -85,B 0,C 180,E1 -1247.016,E2 -1247.016} C_VEL
LIN {X 0,Y 594.39,Z 241.258,A -85,B 0,C 180,E1 -1249.784,E2 -1249.784} C_VEL
LIN {X 0,Y 594.387,Z 241.252,A -85,B 0,C 180,E1 -1252.526,E2 -1252.526} C_VEL
LIN {X 0,Y 594.392,Z 241.257,A -85,B 0,C 180,E1 -1255.252,E2 -1255.252} C_VEL
LIN {X 0,Y 594.39,Z 241.255,A -85,B 0,C 180,E1 -1257.967,E2 -1257.967} C_VEL
LIN {X 0,Y 594.419,Z 241.248,A -85,B 0,C 180,E1 -1260.677,E2 -1260.677} C_VEL
LIN {X 0,Y 594.377,Z 241.261,A -85,B 0,C 180,E1 -1263.389,E2 -1263.389} C_VEL
LIN {X 0,Y 594.363,Z 241.257,A -85,B 0,C 180,E1 -1266.108,E2 -1266.108} C_VEL
LIN {X 0,Y 594.395,Z 241.252,A -85,B 0,C 180,E1 -1268.841,E2 -1268.841} C_VEL
LIN {X 0,Y 594.386,Z 241.262,A -85,B 0,C 180,E1 -1271.595,E2 -1271.595} C_VEL
LIN {X 0,Y 594.381,Z 241.253,A -85,B 0,C 180,E1 -1274.376,E2 -1274.376} C_VEL
LIN {X 0,Y 594.356,Z 241.259,A -85,B 0,C 180,E1 -1275.337,E2 -1275.337} C_VEL
LIN {X 0,Y 593.685,Z 241.346,A -85,B 0,C 180,E1 -1275.903,E2 -1275.903} C_VEL
LIN {X 0,Y 590.831,Z 241.7,A -85,B 0,C 180,E1 -1276.821,E2 -1276.821} C_VEL
LIN {X 0,Y 588.426,Z 242.005,A -85,B 0,C 180,E1 -1277.56,E2 -1277.56} C_VEL
LIN {X 0,Y 587.399,Z 242.125,A -85,B 0,C 180,E1 -1278.13,E2 -1278.13} C_VEL
LIN {X 0,Y 587.319,Z 242.133,A -85,B 0,C 180,E1 -1278.323,E2 -1278.323} C_VEL
LIN {X 0,Y 587.349,Z 242.131,A -85,B 0,C 180,E1 -1281.044,E2 -1281.044} C_VEL
LIN {X 0,Y 587.328,Z 242.135,A -85,B 0,C 180,E1 -1284.006,E2 -1284.006} C_VEL
LIN {X 0,Y 587.354,Z 242.129,A -85,B 0,C 180,E1 -1286.277,E2 -1286.277} C_VEL
LIN {X 0,Y 587.344,Z 242.133,A -85,B 0,C 180,E1 -1289.134,E2 -1289.134} C_VEL
LIN {X 0,Y 587.347,Z 242.135,A -85,B 0,C 180,E1 -1291.838,E2 -1291.838} C_VEL
LIN {X 0,Y 587.351,Z 242.129,A -85,B 0,C 180,E1 -1294.349,E2 -1294.349} C_VEL
LIN {X 0,Y 587.343,Z 242.13,A -85,B 0,C 180,E1 -1296.746,E2 -1296.746} C_VEL
LIN {X 0,Y 587.337,Z 242.137,A -85,B 0,C 180,E1 -1299.359,E2 -1299.359} C_VEL
LIN {X 0,Y 587.324,Z 242.134,A -85,B 0,C 180,E1 -1302.107,E2 -1302.107} C_VEL
LIN {X 0,Y 587.305,Z 242.137,A -85,B 0,C 180,E1 -1305.089,E2 -1305.089} C_VEL
LIN {X 0,Y 587.342,Z 242.134,A -85,B 0,C 180,E1 -1307.927,E2 -1307.927} C_VEL
LIN {X 0,Y 587.325,Z 242.134,A -85,B 0,C 180,E1 -1311.058,E2 -1311.058} C_VEL
LIN {X 0,Y 587.341,Z 242.135,A -85,B 0,C 180,E1 -1313.292,E2 -1313.292} C_VEL
LIN {X 0,Y 587.357,Z 242.134,A -85,B 0,C 180,E1 -1315.78,E2 -1315.78} C_VEL
LIN {X 0,Y 587.346,Z 242.13,A -85,B 0,C 180,E1 -1318.232,E2 -1318.232} C_VEL
LIN {X 0,Y 587.342,Z 242.13,A -85,B 0,C 180,E1 -1320.866,E2 -1320.866} C_VEL
LIN {X 0,Y 587.349,Z 242.135,A -85,B 0,C 180,E1 -1323.819,E2 -1323.819} C_VEL
LIN {X 0,Y 587.355,Z 242.128,A -85,B 0,C 180,E1 -1326.743,E2 -1326.743} C_VEL
LIN {X 0,Y 587.325,Z 242.14,A -85,B 0,C 180,E1 -1329.695,E2 -1329.695} C_VEL
LIN {X 0,Y 587.341,Z 242.13,A -85,B 0,C 180,E1 -1332.594,E2 -1332.594} C_VEL
LIN {X 0,Y 587.355,Z 242.136,A -85,B 0,C 180,E1 -1335.739,E2 -1335.739} C_VEL
LIN {X 0,Y 587.354,Z 242.129,A -85,B 0,C 180,E1 -1338.859,E2 -1338.859} C_VEL
LIN {X 0,Y 587.358,Z 242.135,A -85,B 0,C 180,E1 -1341.745,E2 -1341.745} C_VEL
LIN {X 0,Y 587.341,Z 242.13,A -85,B 0,C 180,E1 -1344.507,E2 -1344.507} C_VEL
LIN {X 0,Y 587.373,Z 242.131,A -85,B 0,C 180,E1 -1347.257,E2 -1347.257} C_VEL
LIN {X 0,Y 587.361,Z 242.131,A -85,B 0,C 180,E1 -1350,E2 -1350} C_VEL
LIN {X 0,Y 587.358,Z 242.128,A -85,B 0,C 180,E1 -1352.743,E2 -1352.743} C_VEL
LIN {X 0,Y 587.35,Z 242.138,A -85,B 0,C 180,E1 -1355.493,E2 -1355.493} C_VEL
LIN {X 0,Y 587.329,Z 242.132,A -85,B 0,C 180,E1 -1358.255,E2 -1358.255} C_VEL
LIN {X 0,Y 587.338,Z 242.133,A -85,B 0,C 180,E1 -1361.133,E2 -1361.133} C_VEL
LIN {X 0,Y 587.342,Z 242.136,A -85,B 0,C 180,E1 -1363.846,E2 -1363.846} C_VEL
LIN {X 0,Y 587.324,Z 242.132,A -85,B 0,C 180,E1 -1366.81,E2 -1366.81} C_VEL
LIN {X 0,Y 587.329,Z 242.142,A -85,B 0,C 180,E1 -1369.575,E2 -1369.575} C_VEL
LIN {X 0,Y 587.322,Z 242.132,A -85,B 0,C 180,E1 -1372.514,E2 -1372.514} C_VEL
LIN {X 0,Y 587.324,Z 242.141,A -85,B 0,C 180,E1 -1375.516,E2 -1375.516} C_VEL
LIN {X 0,Y 587.331,Z 242.138,A -85,B 0,C 180,E1 -1377.818,E2 -1377.818} C_VEL
LIN {X 0,Y 587.313,Z 242.133,A -85,B 0,C 180,E1 -1380.508,E2 -1380.508} C_VEL
LIN {X 0,Y 587.326,Z 242.18,A -85,B 0,C 180,E1 -1383.161,E2 -1383.161} C_VEL
LIN {X 0,Y 587.207,Z 254.051,A -85,B 0,C 180,E1 -1385.905,E2 -1385.905} C_VEL
LIN {X 0,Y 587.206,Z 265.291,A -85,B 0,C 180,E1 -1388.463,E2 -1388.463} C_VEL
LIN {X 0,Y 587.57,Z 271.667,A -85,B 0,C 180,E1 -1388.547,E2 -1388.547} C_VEL
LIN {X 0,Y 587.472,Z 339.61,A -85,B 0,C 180,E1 -1389.39,E2 -1389.39} C_VEL
LIN {X 0,Y 587.399,Z 348.94,A -85,B 0,C 180,E1 -1389.59,E2 -1389.59} C_VEL
LIN {X 0,Y 587.385,Z 358.972,A -85,B 0,C 180,E1 -1389.911,E2 -1389.911} C_VEL
LIN {X 0,Y 587.388,Z 370.239,A -85,B 0,C 180,E1 -1390.416,E2 -1390.416} C_VEL
LIN {X 0,Y 587.338,Z 380.161,A -85,B 0,C 180,E1 -1391.022,E2 -1391.022} C_VEL
LIN {X 0,Y 587.31,Z 387.946,A -85,B 0,C 180,E1 -1391.615,E2 -1391.615} C_VEL
LIN {X 0,Y 587.256,Z 394.162,A -85,B 0,C 180,E1 -1392.184,E2 -1392.184} C_VEL
LIN {X 0,Y 587.249,Z 399.659,A -85,B 0,C 180,E1 -1392.777,E2 -1392.777} C_VEL
LIN {X 0,Y 587.221,Z 405.313,A -85,B 0,C 180,E1 -1393.508,E2 -1393.508} C_VEL
LIN {X 0,Y 587.202,Z 410.159,A -85,B 0,C 180,E1 -1394.27,E2 -1394.27} C_VEL
LIN {X 0,Y 587.176,Z 414.292,A -85,B 0,C 180,E1 -1395.076,E2 -1395.076} C_VEL
LIN {X 0,Y 587.176,Z 417.597,A -85,B 0,C 180,E1 -1395.9,E2 -1395.9} C_VEL
LIN {X 0,Y 587.172,Z 419.516,A -85,B 0,C 180,E1 -1396.493,E2 -1396.493} C_VEL
LIN {X 0,Y 587.16,Z 420.665,A -85,B 0,C 180,E1 -1396.981,E2 -1396.981} C_VEL
LIN {X 0,Y 587.149,Z 422.261,A -85,B 0,C 180,E1 -1397.911,E2 -1397.911} C_VEL
LIN {X 0,Y 587.114,Z 422.98,A -85,B 0,C 180,E1 -1398.948,E2 -1398.948} C_VEL
LIN {X 0,Y 587.14,Z 422.505,A -85,B 0,C 180,E1 -1400.001,E2 -1400.001} C_VEL
LIN {X 0,Y 587.153,Z 420.738,A -85,B 0,C 180,E1 -1401.078,E2 -1401.078} C_VEL
LIN {X 0,Y 587.155,Z 417.62,A -85,B 0,C 180,E1 -1402.183,E2 -1402.183} C_VEL
LIN {X 0,Y 587.214,Z 412.968,A -85,B 0,C 180,E1 -1403.308,E2 -1403.308} C_VEL
LIN {X 0,Y 587.212,Z 407.177,A -85,B 0,C 180,E1 -1404.31,E2 -1404.31} C_VEL
LIN {X 0,Y 587.234,Z 401.138,A -85,B 0,C 180,E1 -1405.134,E2 -1405.134} C_VEL
LIN {X 0,Y 587.271,Z 394.434,A -85,B 0,C 180,E1 -1405.879,E2 -1405.879} C_VEL
LIN {X 0,Y 587.289,Z 386.455,A -85,B 0,C 180,E1 -1406.602,E2 -1406.602} C_VEL
LIN {X 0,Y 587.383,Z 376.11,A -85,B 0,C 180,E1 -1407.334,E2 -1407.334} C_VEL
LIN {X 0,Y 587.404,Z 366.104,A -85,B 0,C 180,E1 -1407.873,E2 -1407.873} C_VEL
LIN {X 0,Y 587.418,Z 357.346,A -85,B 0,C 180,E1 -1408.237,E2 -1408.237} C_VEL
LIN {X 0,Y 587.463,Z 347.809,A -85,B 0,C 180,E1 -1408.529,E2 -1408.529} C_VEL
LIN {X 0,Y 587.496,Z 337.735,A -85,B 0,C 180,E1 -1408.731,E2 -1408.731} C_VEL
LIN {X 0,Y 587.526,Z 267.343,A -85,B 0,C 180,E1 -1409.596,E2 -1409.596} C_VEL
LIN {X 0,Y 587.239,Z 265.212,A -85,B 0,C 180,E1 -1409.629,E2 -1409.629} C_VEL
LIN {X 0,Y 587.28,Z 252.076,A -85,B 0,C 180,E1 -1412.638,E2 -1412.638} C_VEL
LIN {X 0,Y 587.327,Z 242.135,A -85,B 0,C 180,E1 -1414.958,E2 -1414.958} C_VEL
LIN {X 0,Y 587.331,Z 242.132,A -85,B 0,C 180,E1 -1417.487,E2 -1417.487} C_VEL
LIN {X 0,Y 587.324,Z 242.133,A -85,B 0,C 180,E1 -1419.696,E2 -1419.696} C_VEL
LIN {X 0,Y 587.349,Z 242.138,A -85,B 0,C 180,E1 -1422.595,E2 -1422.595} C_VEL
LIN {X 0,Y 587.353,Z 242.129,A -85,B 0,C 180,E1 -1425.74,E2 -1425.74} C_VEL
LIN {X 0,Y 587.351,Z 242.133,A -85,B 0,C 180,E1 -1428.859,E2 -1428.859} C_VEL
LIN {X 0,Y 587.362,Z 242.128,A -85,B 0,C 180,E1 -1431.745,E2 -1431.745} C_VEL
LIN {X 0,Y 587.351,Z 242.139,A -85,B 0,C 180,E1 -1434.508,E2 -1434.508} C_VEL
LIN {X 0,Y 587.374,Z 242.126,A -85,B 0,C 180,E1 -1437.257,E2 -1437.257} C_VEL
LIN {X 0,Y 587.373,Z 242.128,A -85,B 0,C 180,E1 -1440.001,E2 -1440.001} C_VEL
LIN {X 0,Y 587.373,Z 242.132,A -85,B 0,C 180,E1 -1442.744,E2 -1442.744} C_VEL
LIN {X 0,Y 587.351,Z 242.128,A -85,B 0,C 180,E1 -1445.494,E2 -1445.494} C_VEL
LIN {X 0,Y 587.364,Z 242.133,A -85,B 0,C 180,E1 -1448.256,E2 -1448.256} C_VEL
LIN {X 0,Y 587.338,Z 242.131,A -85,B 0,C 180,E1 -1451.134,E2 -1451.134} C_VEL
LIN {X 0,Y 587.35,Z 242.13,A -85,B 0,C 180,E1 -1453.846,E2 -1453.846} C_VEL
LIN {X 0,Y 587.355,Z 242.132,A -85,B 0,C 180,E1 -1456.82,E2 -1456.82} C_VEL
LIN {X 0,Y 587.337,Z 242.13,A -85,B 0,C 180,E1 -1459.576,E2 -1459.576} C_VEL
LIN {X 0,Y 587.317,Z 242.133,A -85,B 0,C 180,E1 -1461.775,E2 -1461.775} C_VEL
LIN {X 0,Y 587.345,Z 242.134,A -85,B 0,C 180,E1 -1464.759,E2 -1464.759} C_VEL
LIN {X 0,Y 587.322,Z 242.134,A -85,B 0,C 180,E1 -1467.047,E2 -1467.047} C_VEL
LIN {X 0,Y 587.346,Z 242.128,A -85,B 0,C 180,E1 -1469.38,E2 -1469.38} C_VEL
LIN {X 0,Y 587.345,Z 242.13,A -85,B 0,C 180,E1 -1471.838,E2 -1471.838} C_VEL
LIN {X 0,Y 587.348,Z 242.136,A -85,B 0,C 180,E1 -1474.35,E2 -1474.35} C_VEL
LIN {X 0,Y 587.346,Z 242.135,A -85,B 0,C 180,E1 -1476.747,E2 -1476.747} C_VEL
LIN {X 0,Y 587.34,Z 242.13,A -85,B 0,C 180,E1 -1479.36,E2 -1479.36} C_VEL
LIN {X 0,Y 587.329,Z 242.135,A -85,B 0,C 180,E1 -1482.109,E2 -1482.109} C_VEL
LIN {X 0,Y 587.311,Z 242.135,A -85,B 0,C 180,E1 -1485.09,E2 -1485.09} C_VEL
LIN {X 0,Y 587.349,Z 242.131,A -85,B 0,C 180,E1 -1487.928,E2 -1487.928} C_VEL
LIN {X 0,Y 587.318,Z 242.135,A -85,B 0,C 180,E1 -1491.06,E2 -1491.06} C_VEL
LIN {X 0,Y 587.349,Z 242.129,A -85,B 0,C 180,E1 -1493.293,E2 -1493.293} C_VEL
LIN {X 0,Y 587.357,Z 242.129,A -85,B 0,C 180,E1 -1495.781,E2 -1495.781} C_VEL
LIN {X 0,Y 587.338,Z 242.136,A -85,B 0,C 180,E1 -1498.232,E2 -1498.232} C_VEL
LIN {X 0,Y 587.343,Z 242.134,A -85,B 0,C 180,E1 -1500.868,E2 -1500.868} C_VEL
LIN {X 0,Y 587.33,Z 242.133,A -85,B 0,C 180,E1 -1503.825,E2 -1503.825} C_VEL
LIN {X 0,Y 587.335,Z 242.134,A -85,B 0,C 180,E1 -1505.994,E2 -1505.994} C_VEL
LIN {X 0,Y 587.355,Z 242.231,A -85,B 0,C 180,E1 -1507.286,E2 -1507.286} C_VEL
LIN {X 0,Y 587.742,Z 245.894,A -85,B 0,C 180,E1 -1507.873,E2 -1507.873} C_VEL
LIN {X 0,Y 587.624,Z 261.322,A -85,B 0,C 180,E1 -1510.253,E2 -1510.253} C_VEL
LIN {X 0,Y 587.474,Z 278.922,A -85,B 0,C 180,E1 -1512.926,E2 -1512.926} C_VEL
LIN {X 0,Y 587.418,Z 297.557,A -85,B 0,C 180,E1 -1515.72,E2 -1515.72} C_VEL
LIN {X 0,Y 587.335,Z 316.035,A -85,B 0,C 180,E1 -1518.456,E2 -1518.456} C_VEL
LIN {X 0,Y 587.275,Z 322.325,A -85,B 0,C 180,E1 -1519.38,E2 -1519.38} C_VEL
LIN {X 0,Y 587.586,Z 329.152,A -85,B 0,C 180,E1 -1519.472,E2 -1519.472} C_VEL
LIN {X 0,Y 587.514,Z 399.161,A -85,B 0,C 180,E1 -1520.338,E2 -1520.338} C_VEL
LIN {X 0,Y 587.453,Z 408.428,A -85,B 0,C 180,E1 -1520.532,E2 -1520.532} C_VEL
LIN {X 0,Y 587.416,Z 416.902,A -85,B 0,C 180,E1 -1520.792,E2 -1520.792} C_VEL
LIN {X 0,Y 587.367,Z 425.406,A -85,B 0,C 180,E1 -1521.138,E2 -1521.138} C_VEL
LIN {X 0,Y 587.393,Z 433.734,A -85,B 0,C 180,E1 -1521.572,E2 -1521.572} C_VEL
LIN {X 0,Y 587.332,Z 441.77,A -85,B 0,C 180,E1 -1522.091,E2 -1522.091} C_VEL
LIN {X 0,Y 587.288,Z 449.42,A -85,B 0,C 180,E1 -1522.696,E2 -1522.696} C_VEL
LIN {X 0,Y 587.281,Z 457.811,A -85,B 0,C 180,E1 -1523.512,E2 -1523.512} C_VEL
LIN {X 0,Y 587.238,Z 464.434,A -85,B 0,C 180,E1 -1524.334,E2 -1524.334} C_VEL
LIN {X 0,Y 587.17,Z 469.988,A -85,B 0,C 180,E1 -1525.194,E2 -1525.194} C_VEL
LIN {X 0,Y 587.211,Z 475.148,A -85,B 0,C 180,E1 -1526.226,E2 -1526.226} C_VEL
LIN {X 0,Y 587.155,Z 477.789,A -85,B 0,C 180,E1 -1526.913,E2 -1526.913} C_VEL
LIN {X 0,Y 587.141,Z 480.681,A -85,B 0,C 180,E1 -1527.942,E2 -1527.942} C_VEL
LIN {X 0,Y 587.145,Z 481.936,A -85,B 0,C 180,E1 -1528.628,E2 -1528.628} C_VEL
LIN {X 0,Y 587.136,Z 482.712,A -85,B 0,C 180,E1 -1529.314,E2 -1529.314} C_VEL
LIN {X 0,Y 587.134,Z 483,A -85,B 0,C 180,E1 -1530,E2 -1530} C_VEL
LIN {X 0,Y 587.136,Z 482.711,A -85,B 0,C 180,E1 -1530.686,E2 -1530.686} C_VEL
LIN {X 0,Y 587.145,Z 481.936,A -85,B 0,C 180,E1 -1531.372,E2 -1531.372} C_VEL
LIN {X 0,Y 587.141,Z 480.68,A -85,B 0,C 180,E1 -1532.058,E2 -1532.058} C_VEL
LIN {X 0,Y 587.155,Z 477.787,A -85,B 0,C 180,E1 -1533.088,E2 -1533.088} C_VEL
LIN {X 0,Y 587.211,Z 475.147,A -85,B 0,C 180,E1 -1533.774,E2 -1533.774} C_VEL
LIN {X 0,Y 587.17,Z 469.985,A -85,B 0,C 180,E1 -1534.806,E2 -1534.806} C_VEL
LIN {X 0,Y 587.253,Z 463.187,A -85,B 0,C 180,E1 -1535.839,E2 -1535.839} C_VEL
LIN {X 0,Y 587.269,Z 456.287,A -85,B 0,C 180,E1 -1536.645,E2 -1536.645} C_VEL
LIN {X 0,Y 587.292,Z 448.405,A -85,B 0,C 180,E1 -1537.391,E2 -1537.391} C_VEL
LIN {X 0,Y 587.339,Z 440.549,A -85,B 0,C 180,E1 -1537.996,E2 -1537.996} C_VEL
LIN {X 0,Y 587.38,Z 430.734,A -85,B 0,C 180,E1 -1538.602,E2 -1538.602} C_VEL
LIN {X 0,Y 587.42,Z 419.3,A -85,B 0,C 180,E1 -1539.121,E2 -1539.121} C_VEL
LIN {X 0,Y 587.451,Z 409.246,A -85,B 0,C 180,E1 -1539.446,E2 -1539.446} C_VEL
LIN {X 0,Y 587.484,Z 400.446,A -85,B 0,C 180,E1 -1539.641,E2 -1539.641} C_VEL
LIN {X 0,Y 587.581,Z 327.371,A -85,B 0,C 180,E1 -1540.55,E2 -1540.55} C_VEL
LIN {X 0,Y 587.275,Z 322.324,A -85,B 0,C 180,E1 -1540.62,E2 -1540.62} C_VEL
LIN {X 0,Y 587.4,Z 304.046,A -85,B 0,C 180,E1 -1543.316,E2 -1543.316} C_VEL
LIN {X 0,Y 587.488,Z 283.87,A -85,B 0,C 180,E1 -1546.327,E2 -1546.327} C_VEL
LIN {X 0,Y 587.591,Z 264.406,A -85,B 0,C 180,E1 -1549.275,E2 -1549.275} C_VEL
LIN {X 0,Y 587.752,Z 248.265,A -85,B 0,C 180,E1 -1551.757,E2 -1551.757} C_VEL
LIN {X 0,Y 587.586,Z 243.518,A -85,B 0,C 180,E1 -1552.504,E2 -1552.504} C_VEL
LIN {X 0,Y 587.338,Z 242.136,A -85,B 0,C 180,E1 -1552.739,E2 -1552.739} C_VEL
LIN {X 0,Y 587.333,Z 242.141,A -85,B 0,C 180,E1 -1555.516,E2 -1555.516} C_VEL
LIN {X 0,Y 587.337,Z 242.136,A -85,B 0,C 180,E1 -1557.818,E2 -1557.818} C_VEL
LIN {X 0,Y 587.334,Z 242.13,A -85,B 0,C 180,E1 -1560.509,E2 -1560.509} C_VEL
LIN {X 0,Y 587.335,Z 242.139,A -85,B 0,C 180,E1 -1563.396,E2 -1563.396} C_VEL
LIN {X 0,Y 587.302,Z 242.139,A -85,B 0,C 180,E1 -1565.899,E2 -1565.899} C_VEL
LIN {X 0,Y 587.32,Z 242.132,A -85,B 0,C 180,E1 -1568.479,E2 -1568.479} C_VEL
LIN {X 0,Y 587.333,Z 242.135,A -85,B 0,C 180,E1 -1571.156,E2 -1571.156} C_VEL
LIN {X 0,Y 587.324,Z 242.133,A -85,B 0,C 180,E1 -1574.113,E2 -1574.113} C_VEL
LIN {X 0,Y 587.309,Z 242.136,A -85,B 0,C 180,E1 -1576.993,E2 -1576.993} C_VEL
LIN {X 0,Y 587.315,Z 242.14,A -85,B 0,C 180,E1 -1579.745,E2 -1579.745} C_VEL
LIN {X 0,Y 587.34,Z 242.13,A -85,B 0,C 180,E1 -1582.392,E2 -1582.392} C_VEL
LIN {X 0,Y 587.322,Z 242.134,A -85,B 0,C 180,E1 -1584.944,E2 -1584.944} C_VEL
LIN {X 0,Y 587.336,Z 242.139,A -85,B 0,C 180,E1 -1587.421,E2 -1587.421} C_VEL
LIN {X 0,Y 587.329,Z 242.137,A -85,B 0,C 180,E1 -1589.829,E2 -1589.829} C_VEL
LIN {X 0,Y 587.347,Z 242.129,A -85,B 0,C 180,E1 -1592.306,E2 -1592.306} C_VEL
LIN {X 0,Y 587.335,Z 242.13,A -85,B 0,C 180,E1 -1594.483,E2 -1594.483} C_VEL
LIN {X 0,Y 587.335,Z 242.14,A -85,B 0,C 180,E1 -1597.486,E2 -1597.486} C_VEL
LIN {X 0,Y 587.339,Z 242.13,A -85,B 0,C 180,E1 -1600.424,E2 -1600.424} C_VEL
LIN {X 0,Y 587.348,Z 242.135,A -85,B 0,C 180,E1 -1603.311,E2 -1603.311} C_VEL
LIN {X 0,Y 587.352,Z 242.13,A -85,B 0,C 180,E1 -1606.154,E2 -1606.154} C_VEL
LIN {X 0,Y 587.337,Z 242.132,A -85,B 0,C 180,E1 -1608.962,E2 -1608.962} C_VEL
LIN {X 0,Y 587.365,Z 242.134,A -85,B 0,C 180,E1 -1611.744,E2 -1611.744} C_VEL
LIN {X 0,Y 587.351,Z 242.128,A -85,B 0,C 180,E1 -1614.506,E2 -1614.506} C_VEL
LIN {X 0,Y 587.372,Z 242.131,A -85,B 0,C 180,E1 -1617.256,E2 -1617.256} C_VEL
LIN {X 0,Y 587.376,Z 242.129,A -85,B 0,C 180,E1 -1619.999,E2 -1619.999} C_VEL
LIN {X 0,Y 587.375,Z 242.126,A -85,B 0,C 180,E1 -1622.743,E2 -1622.743} C_VEL
LIN {X 0,Y 587.349,Z 242.138,A -85,B 0,C 180,E1 -1625.492,E2 -1625.492} C_VEL
LIN {X 0,Y 587.365,Z 242.128,A -85,B 0,C 180,E1 -1628.255,E2 -1628.255} C_VEL
LIN {X 0,Y 587.339,Z 242.134,A -85,B 0,C 180,E1 -1631.133,E2 -1631.133} C_VEL
LIN {X 0,Y 587.351,Z 242.134,A -85,B 0,C 180,E1 -1633.845,E2 -1633.845} C_VEL
LIN {X 0,Y 587.353,Z 242.129,A -85,B 0,C 180,E1 -1636.819,E2 -1636.819} C_VEL
LIN {X 0,Y 587.319,Z 242.133,A -85,B 0,C 180,E1 -1638.323,E2 -1638.323} C_VEL
LIN {X 0,Y 586.667,Z 242.215,A -85,B 0,C 180,E1 -1638.895,E2 -1638.895} C_VEL
LIN {X 0,Y 583.837,Z 242.573,A -85,B 0,C 180,E1 -1639.823,E2 -1639.823} C_VEL
LIN {X 0,Y 581.427,Z 242.876,A -85,B 0,C 180,E1 -1640.57,E2 -1640.57} C_VEL
LIN {X 0,Y 580.374,Z 243.005,A -85,B 0,C 180,E1 -1641.146,E2 -1641.146} C_VEL
LIN {X 0,Y 580.279,Z 243.015,A -85,B 0,C 180,E1 -1641.342,E2 -1641.342} C_VEL
LIN {X 0,Y 580.291,Z 243.008,A -85,B 0,C 180,E1 -1644.316,E2 -1644.316} C_VEL
LIN {X 0,Y 580.298,Z 243.007,A -85,B 0,C 180,E1 -1646.621,E2 -1646.621} C_VEL
LIN {X 0,Y 580.295,Z 243.014,A -85,B 0,C 180,E1 -1649.31,E2 -1649.31} C_VEL
LIN {X 0,Y 580.294,Z 243.009,A -85,B 0,C 180,E1 -1652.2,E2 -1652.2} C_VEL
LIN {X 0,Y 580.294,Z 243.008,A -85,B 0,C 180,E1 -1654.695,E2 -1654.695} C_VEL
LIN {X 0,Y 580.29,Z 243.014,A -85,B 0,C 180,E1 -1657.268,E2 -1657.268} C_VEL
LIN {X 0,Y 580.288,Z 243.009,A -85,B 0,C 180,E1 -1660.271,E2 -1660.271} C_VEL
LIN {X 0,Y 580.271,Z 243.011,A -85,B 0,C 180,E1 -1662.706,E2 -1662.706} C_VEL
LIN {X 0,Y 580.263,Z 243.021,A -85,B 0,C 180,E1 -1665.608,E2 -1665.608} C_VEL
LIN {X 0,Y 580.304,Z 243.007,A -85,B 0,C 180,E1 -1668.234,E2 -1668.234} C_VEL
LIN {X 0,Y 580.28,Z 243.011,A -85,B 0,C 180,E1 -1670.966,E2 -1670.966} C_VEL
LIN {X 0,Y 580.267,Z 243.021,A -85,B 0,C 180,E1 -1673.597,E2 -1673.597} C_VEL
LIN {X 0,Y 580.309,Z 243.008,A -85,B 0,C 180,E1 -1676.145,E2 -1676.145} C_VEL
LIN {X 0,Y 580.28,Z 243.009,A -85,B 0,C 180,E1 -1678.615,E2 -1678.615} C_VEL
LIN {X 0,Y 580.287,Z 243.011,A -85,B 0,C 180,E1 -1681.024,E2 -1681.024} C_VEL
LIN {X 0,Y 580.282,Z 243.018,A -85,B 0,C 180,E1 -1683.666,E2 -1683.666} C_VEL
LIN {X 0,Y 580.29,Z 243.008,A -85,B 0,C 180,E1 -1686.443,E2 -1686.443} C_VEL
LIN {X 0,Y 580.275,Z 243.018,A -85,B 0,C 180,E1 -1689.437,E2 -1689.437} C_VEL
LIN {X 0,Y 580.26,Z 243.021,A -85,B 0,C 180,E1 -1691.645,E2 -1691.645} C_VEL
LIN {X 0,Y 580.272,Z 243.016,A -85,B 0,C 180,E1 -1693.826,E2 -1693.826} C_VEL
LIN {X 0,Y 580.315,Z 243.009,A -85,B 0,C 180,E1 -1695.983,E2 -1695.983} C_VEL
LIN {X 0,Y 580.323,Z 243.005,A -85,B 0,C 180,E1 -1698.827,E2 -1698.827} C_VEL
LIN {X 0,Y 580.323,Z 243.014,A -85,B 0,C 180,E1 -1701.644,E2 -1701.644} C_VEL
LIN {X 0,Y 580.307,Z 243.006,A -85,B 0,C 180,E1 -1704.44,E2 -1704.44} C_VEL
LIN {X 0,Y 580.338,Z 243.007,A -85,B 0,C 180,E1 -1707.223,E2 -1707.223} C_VEL
LIN {X 0,Y 580.331,Z 243.007,A -85,B 0,C 180,E1 -1710,E2 -1710} C_VEL
LIN {X 0,Y 580.326,Z 243.004,A -85,B 0,C 180,E1 -1712.776,E2 -1712.776} C_VEL
LIN {X 0,Y 580.313,Z 243.015,A -85,B 0,C 180,E1 -1715.56,E2 -1715.56} C_VEL
LIN {X 0,Y 580.299,Z 243.008,A -85,B 0,C 180,E1 -1718.356,E2 -1718.356} C_VEL
LIN {X 0,Y 580.29,Z 243.012,A -85,B 0,C 180,E1 -1721.191,E2 -1721.191} C_VEL
LIN {X 0,Y 580.298,Z 243.011,A -85,B 0,C 180,E1 -1724.017,E2 -1724.017} C_VEL
LIN {X 0,Y 580.301,Z 243.008,A -85,B 0,C 180,E1 -1726.914,E2 -1726.914} C_VEL
LIN {X 0,Y 580.289,Z 243.015,A -85,B 0,C 180,E1 -1729.822,E2 -1729.822} C_VEL
LIN {X 0,Y 580.28,Z 243.01,A -85,B 0,C 180,E1 -1732.802,E2 -1732.802} C_VEL
LIN {X 0,Y 580.279,Z 243.012,A -85,B 0,C 180,E1 -1735.08,E2 -1735.08} C_VEL
LIN {X 0,Y 580.282,Z 243.011,A -85,B 0,C 180,E1 -1738.186,E2 -1738.186} C_VEL
LIN {X 0,Y 580.267,Z 243.011,A -85,B 0,C 180,E1 -1740.694,E2 -1740.694} C_VEL
LIN {X 0,Y 580.277,Z 243.052,A -85,B 0,C 180,E1 -1743.168,E2 -1743.168} C_VEL
LIN {X 0,Y 580.147,Z 255.372,A -85,B 0,C 180,E1 -1746.05,E2 -1746.05} C_VEL
LIN {X 0,Y 580.105,Z 265.194,A -85,B 0,C 180,E1 -1748.325,E2 -1748.325} C_VEL
LIN {X 0,Y 580.604,Z 270.919,A -85,B 0,C 180,E1 -1748.411,E2 -1748.411} C_VEL
LIN {X 0,Y 580.484,Z 339.966,A -85,B 0,C 180,E1 -1749.278,E2 -1749.278} C_VEL
LIN {X 0,Y 580.427,Z 349.738,A -85,B 0,C 180,E1 -1749.496,E2 -1749.496} C_VEL
LIN {X 0,Y 580.361,Z 360.956,A -85,B 0,C 180,E1 -1749.873,E2 -1749.873} C_VEL
LIN {X 0,Y 580.346,Z 371.033,A -85,B 0,C 180,E1 -1750.356,E2 -1750.356} C_VEL
LIN {X 0,Y 580.304,Z 380.701,A -85,B 0,C 180,E1 -1750.963,E2 -1750.963} C_VEL
LIN {X 0,Y 580.258,Z 387.649,A -85,B 0,C 180,E1 -1751.499,E2 -1751.499} C_VEL
LIN {X 0,Y 580.183,Z 395.447,A -85,B 0,C 180,E1 -1752.232,E2 -1752.232} C_VEL
LIN {X 0,Y 580.151,Z 402.481,A -85,B 0,C 180,E1 -1753.047,E2 -1753.047} C_VEL
LIN {X 0,Y 580.127,Z 409.125,A -85,B 0,C 180,E1 -1754.024,E2 -1754.024} C_VEL
LIN {X 0,Y 580.092,Z 414.155,A -85,B 0,C 180,E1 -1754.996,E2 -1754.996} C_VEL
LIN {X 0,Y 580.083,Z 417.975,A -85,B 0,C 180,E1 -1755.976,E2 -1755.976} C_VEL
LIN {X 0,Y 580.059,Z 419.913,A -85,B 0,C 180,E1 -1756.631,E2 -1756.631} C_VEL
LIN {X 0,Y 580.052,Z 421.929,A -85,B 0,C 180,E1 -1757.652,E2 -1757.652} C_VEL
LIN {X 0,Y 580.037,Z 422.638,A -85,B 0,C 180,E1 -1758.211,E2 -1758.211} C_VEL
LIN {X 0,Y 580.01,Z 422.984,A -85,B 0,C 180,E1 -1759.133,E2 -1759.133} C_VEL
LIN {X 0,Y 580.047,Z 422.458,A -85,B 0,C 180,E1 -1760.048,E2 -1760.048} C_VEL
LIN {X 0,Y 580.056,Z 421.095,A -85,B 0,C 180,E1 -1760.948,E2 -1760.948} C_VEL
LIN {X 0,Y 580.082,Z 418.51,A -85,B 0,C 180,E1 -1761.952,E2 -1761.952} C_VEL
LIN {X 0,Y 580.103,Z 414.172,A -85,B 0,C 180,E1 -1763.09,E2 -1763.09} C_VEL
LIN {X 0,Y 580.106,Z 409.781,A -85,B 0,C 180,E1 -1763.947,E2 -1763.947} C_VEL
LIN {X 0,Y 580.16,Z 403.802,A -85,B 0,C 180,E1 -1764.873,E2 -1764.873} C_VEL
LIN {X 0,Y 580.217,Z 395.759,A -85,B 0,C 180,E1 -1765.826,E2 -1765.826} C_VEL
LIN {X 0,Y 580.236,Z 389.351,A -85,B 0,C 180,E1 -1766.445,E2 -1766.445} C_VEL
LIN {X 0,Y 580.306,Z 381.355,A -85,B 0,C 180,E1 -1767.081,E2 -1767.081} C_VEL
LIN {X 0,Y 580.372,Z 373.319,A -85,B 0,C 180,E1 -1767.6,E2 -1767.6} C_VEL
LIN {X 0,Y 580.383,Z 364.213,A -85,B 0,C 180,E1 -1768.07,E2 -1768.07} C_VEL
LIN {X 0,Y 580.456,Z 353.879,A -85,B 0,C 180,E1 -1768.474,E2 -1768.474} C_VEL
LIN {X 0,Y 580.478,Z 341.816,A -85,B 0,C 180,E1 -1768.781,E2 -1768.781} C_VEL
LIN {X 0,Y 580.523,Z 318.18,A -85,B 0,C 180,E1 -1769.099,E2 -1769.099} C_VEL
LIN {X 0,Y 580.543,Z 267.963,A -85,B 0,C 180,E1 -1769.717,E2 -1769.717} C_VEL
LIN {X 0,Y 580.172,Z 265.162,A -85,B 0,C 180,E1 -1769.771,E2 -1769.771} C_VEL
LIN {X 0,Y 580.211,Z 252.983,A -85,B 0,C 180,E1 -1772.595,E2 -1772.595} C_VEL
LIN {X 0,Y 580.282,Z 243.013,A -85,B 0,C 180,E1 -1774.973,E2 -1774.973} C_VEL
LIN {X 0,Y 580.265,Z 243.014,A -85,B 0,C 180,E1 -1777.948,E2 -1777.948} C_VEL
LIN {X 0,Y 580.306,Z 243.011,A -85,B 0,C 180,E1 -1780.914,E2 -1780.914} C_VEL
LIN {X 0,Y 580.272,Z 243.012,A -85,B 0,C 180,E1 -1783.826,E2 -1783.826} C_VEL
LIN {X 0,Y 580.314,Z 243.008,A -85,B 0,C 180,E1 -1785.984,E2 -1785.984} C_VEL
LIN {X 0,Y 580.32,Z 243.009,A -85,B 0,C 180,E1 -1788.828,E2 -1788.828} C_VEL
LIN {X 0,Y 580.326,Z 243.004,A -85,B 0,C 180,E1 -1791.645,E2 -1791.645} C_VEL
LIN {X 0,Y 580.317,Z 243.015,A -85,B 0,C 180,E1 -1794.441,E2 -1794.441} C_VEL
LIN {X 0,Y 580.339,Z 243.002,A -85,B 0,C 180,E1 -1797.224,E2 -1797.224} C_VEL
LIN {X 0,Y 580.342,Z 243.004,A -85,B 0,C 180,E1 -1800.001,E2 -1800.001} C_VEL
LIN {X 0,Y 580.338,Z 243.008,A -85,B 0,C 180,E1 -1802.777,E2 -1802.777} C_VEL
LIN {X 0,Y 580.317,Z 243.005,A -85,B 0,C 180,E1 -1805.56,E2 -1805.56} C_VEL
LIN {X 0,Y 580.327,Z 243.011,A -85,B 0,C 180,E1 -1808.357,E2 -1808.357} C_VEL
LIN {X 0,Y 580.29,Z 243.009,A -85,B 0,C 180,E1 -1811.192,E2 -1811.192} C_VEL
LIN {X 0,Y 580.317,Z 243.007,A -85,B 0,C 180,E1 -1814.018,E2 -1814.018} C_VEL
LIN {X 0,Y 580.305,Z 243.009,A -85,B 0,C 180,E1 -1816.915,E2 -1816.915} C_VEL
LIN {X 0,Y 580.3,Z 243.008,A -85,B 0,C 180,E1 -1819.823,E2 -1819.823} C_VEL
LIN {X 0,Y 580.267,Z 243.014,A -85,B 0,C 180,E1 -1822.053,E2 -1822.053} C_VEL
LIN {X 0,Y 580.302,Z 243.007,A -85,B 0,C 180,E1 -1825.08,E2 -1825.08} C_VEL
LIN {X 0,Y 580.313,Z 243.007,A -85,B 0,C 180,E1 -1827.864,E2 -1827.864} C_VEL
LIN {X 0,Y 580.284,Z 243.016,A -85,B 0,C 180,E1 -1830.697,E2 -1830.697} C_VEL
LIN {X 0,Y 580.298,Z 243.006,A -85,B 0,C 180,E1 -1833.318,E2 -1833.318} C_VEL
LIN {X 0,Y 580.319,Z 243.005,A -85,B 0,C 180,E1 -1835.768,E2 -1835.768} C_VEL
LIN {X 0,Y 580.283,Z 243.013,A -85,B 0,C 180,E1 -1838.147,E2 -1838.147} C_VEL
LIN {X 0,Y 580.293,Z 243.012,A -85,B 0,C 180,E1 -1840.844,E2 -1840.844} C_VEL
LIN {X 0,Y 580.273,Z 243.01,A -85,B 0,C 180,E1 -1843.659,E2 -1843.659} C_VEL
LIN {X 0,Y 580.272,Z 243.019,A -85,B 0,C 180,E1 -1846.61,E2 -1846.61} C_VEL
LIN {X 0,Y 580.293,Z 243.009,A -85,B 0,C 180,E1 -1849.157,E2 -1849.157} C_VEL
LIN {X 0,Y 580.287,Z 243.011,A -85,B 0,C 180,E1 -1851.928,E2 -1851.928} C_VEL
LIN {X 0,Y 580.281,Z 243.02,A -85,B 0,C 180,E1 -1854.456,E2 -1854.456} C_VEL
LIN {X 0,Y 580.288,Z 243.011,A -85,B 0,C 180,E1 -1856.976,E2 -1856.976} C_VEL
LIN {X 0,Y 580.292,Z 243.008,A -85,B 0,C 180,E1 -1859.426,E2 -1859.426} C_VEL
LIN {X 0,Y 580.288,Z 243.014,A -85,B 0,C 180,E1 -1862.144,E2 -1862.144} C_VEL
LIN {X 0,Y 580.32,Z 243.006,A -85,B 0,C 180,E1 -1865.27,E2 -1865.27} C_VEL
LIN {X 0,Y 580.297,Z 243.137,A -85,B 0,C 180,E1 -1867.198,E2 -1867.198} C_VEL
LIN {X 0,Y 580.773,Z 246.887,A -85,B 0,C 180,E1 -1867.781,E2 -1867.781} C_VEL
LIN {X 0,Y 580.66,Z 262.509,A -85,B 0,C 180,E1 -1870.191,E2 -1870.191} C_VEL
LIN {X 0,Y 580.482,Z 279.362,A -85,B 0,C 180,E1 -1872.782,E2 -1872.782} C_VEL
LIN {X 0,Y 580.392,Z 295.74,A -85,B 0,C 180,E1 -1875.269,E2 -1875.269} C_VEL
LIN {X 0,Y 580.317,Z 314.73,A -85,B 0,C 180,E1 -1878.119,E2 -1878.119} C_VEL
LIN {X 0,Y 580.211,Z 322.281,A -85,B 0,C 180,E1 -1879.243,E2 -1879.243} C_VEL
LIN {X 0,Y 580.613,Z 327.828,A -85,B 0,C 180,E1 -1879.328,E2 -1879.328} C_VEL
LIN {X 0,Y 580.54,Z 399.161,A -85,B 0,C 180,E1 -1880.221,E2 -1880.221} C_VEL
LIN {X 0,Y 580.467,Z 408.427,A -85,B 0,C 180,E1 -1880.417,E2 -1880.417} C_VEL
LIN {X 0,Y 580.423,Z 416.902,A -85,B 0,C 180,E1 -1880.68,E2 -1880.68} C_VEL
LIN {X 0,Y 580.363,Z 425.408,A -85,B 0,C 180,E1 -1881.031,E2 -1881.031} C_VEL
LIN {X 0,Y 580.348,Z 433.737,A -85,B 0,C 180,E1 -1881.469,E2 -1881.469} C_VEL
LIN {X 0,Y 580.309,Z 441.772,A -85,B 0,C 180,E1 -1881.994,E2 -1881.994} C_VEL
LIN {X 0,Y 580.223,Z 450.434,A -85,B 0,C 180,E1 -1882.694,E2 -1882.694} C_VEL
LIN {X 0,Y 580.218,Z 458.42,A -85,B 0,C 180,E1 -1883.504,E2 -1883.504} C_VEL
LIN {X 0,Y 580.173,Z 464.435,A -85,B 0,C 180,E1 -1884.265,E2 -1884.265} C_VEL
LIN {X 0,Y 580.084,Z 469.989,A -85,B 0,C 180,E1 -1885.135,E2 -1885.135} C_VEL
LIN {X 0,Y 580.137,Z 475.149,A -85,B 0,C 180,E1 -1886.18,E2 -1886.18} C_VEL
LIN {X 0,Y 580.07,Z 477.789,A -85,B 0,C 180,E1 -1886.875,E2 -1886.875} C_VEL
LIN {X 0,Y 580.04,Z 480.682,A -85,B 0,C 180,E1 -1887.917,E2 -1887.917} C_VEL
LIN {X 0,Y 580.045,Z 481.936,A -85,B 0,C 180,E1 -1888.612,E2 -1888.612} C_VEL
LIN {X 0,Y 580.036,Z 482.711,A -85,B 0,C 180,E1 -1889.306,E2 -1889.306} C_VEL
LIN {X 0,Y 580.034,Z 483,A -85,B 0,C 180,E1 -1890,E2 -1890} C_VEL
LIN {X 0,Y 580.036,Z 482.71,A -85,B 0,C 180,E1 -1890.694,E2 -1890.694} C_VEL
LIN {X 0,Y 580.045,Z 481.935,A -85,B 0,C 180,E1 -1891.389,E2 -1891.389} C_VEL
LIN {X 0,Y 580.04,Z 480.68,A -85,B 0,C 180,E1 -1892.083,E2 -1892.083} C_VEL
LIN {X 0,Y 580.07,Z 477.788,A -85,B 0,C 180,E1 -1893.125,E2 -1893.125} C_VEL
LIN {X 0,Y 580.137,Z 475.147,A -85,B 0,C 180,E1 -1893.82,E2 -1893.82} C_VEL
LIN {X 0,Y 580.084,Z 469.985,A -85,B 0,C 180,E1 -1894.865,E2 -1894.865} C_VEL
LIN {X 0,Y 580.193,Z 463.186,A -85,B 0,C 180,E1 -1895.91,E2 -1895.91} C_VEL
LIN {X 0,Y 580.225,Z 455.497,A -85,B 0,C 180,E1 -1896.808,E2 -1896.808} C_VEL
LIN {X 0,Y 580.25,Z 448.406,A -85,B 0,C 180,E1 -1897.481,E2 -1897.481} C_VEL
LIN {X 0,Y 580.299,Z 440.546,A -85,B 0,C 180,E1 -1898.094,E2 -1898.094} C_VEL
LIN {X 0,Y 580.35,Z 430.732,A -85,B 0,C 180,E1 -1898.707,E2 -1898.707} C_VEL
LIN {X 0,Y 580.4,Z 419.302,A -85,B 0,C 180,E1 -1899.233,E2 -1899.233} C_VEL
LIN {X 0,Y 580.465,Z 409.247,A -85,B 0,C 180,E1 -1899.561,E2 -1899.561} C_VEL
LIN {X 0,Y 580.51,Z 400.444,A -85,B 0,C 180,E1 -1899.758,E2 -1899.758} C_VEL
LIN {X 0,Y 580.613,Z 327.784,A -85,B 0,C 180,E1 -1900.673,E2 -1900.673} C_VEL
LIN {X 0,Y 580.209,Z 322.277,A -85,B 0,C 180,E1 -1900.758,E2 -1900.758} C_VEL
LIN {X 0,Y 580.348,Z 305.233,A -85,B 0,C 180,E1 -1903.302,E2 -1903.302} C_VEL
LIN {X 0,Y 580.498,Z 285.057,A -85,B 0,C 180,E1 -1906.349,E2 -1906.349} C_VEL
LIN {X 0,Y 580.597,Z 266.225,A -85,B 0,C 180,E1 -1909.235,E2 -1909.235} C_VEL
LIN {X 0,Y 580.728,Z 253.012,A -85,B 0,C 180,E1 -1911.288,E2 -1911.288} C_VEL
LIN {X 0,Y 580.787,Z 245.74,A -85,B 0,C 180,E1 -1912.406,E2 -1912.406} C_VEL
LIN {X 0,Y 580.288,Z 243.016,A -85,B 0,C 180,E1 -1912.863,E2 -1912.863} C_VEL
LIN {X 0,Y 580.306,Z 243.011,A -85,B 0,C 180,E1 -1915.079,E2 -1915.079} C_VEL
LIN {X 0,Y 580.292,Z 243.009,A -85,B 0,C 180,E1 -1918.186,E2 -1918.186} C_VEL
LIN {X 0,Y 580.281,Z 243.009,A -85,B 0,C 180,E1 -1920.694,E2 -1920.694} C_VEL
LIN {X 0,Y 580.303,Z 243.013,A -85,B 0,C 180,E1 -1923.316,E2 -1923.316} C_VEL
LIN {X 0,Y 580.264,Z 243.018,A -85,B 0,C 180,E1 -1925.758,E2 -1925.758} C_VEL
LIN {X 0,Y 580.284,Z 243.01,A -85,B 0,C 180,E1 -1928.146,E2 -1928.146} C_VEL
LIN {X 0,Y 580.295,Z 243.008,A -85,B 0,C 180,E1 -1930.843,E2 -1930.843} C_VEL
LIN {X 0,Y 580.276,Z 243.018,A -85,B 0,C 180,E1 -1933.657,E2 -1933.657} C_VEL
LIN {X 0,Y 580.273,Z 243.01,A -85,B 0,C 180,E1 -1936.609,E2 -1936.609} C_VEL
LIN {X 0,Y 580.294,Z 243.012,A -85,B 0,C 180,E1 -1939.156,E2 -1939.156} C_VEL
LIN {X 0,Y 580.286,Z 243.012,A -85,B 0,C 180,E1 -1941.926,E2 -1941.926} C_VEL
LIN {X 0,Y 580.282,Z 243.009,A -85,B 0,C 180,E1 -1944.455,E2 -1944.455} C_VEL
LIN {X 0,Y 580.288,Z 243.01,A -85,B 0,C 180,E1 -1946.975,E2 -1946.975} C_VEL
LIN {X 0,Y 580.29,Z 243.017,A -85,B 0,C 180,E1 -1949.424,E2 -1949.424} C_VEL
LIN {X 0,Y 580.316,Z 243.006,A -85,B 0,C 180,E1 -1952.136,E2 -1952.136} C_VEL
LIN {X 0,Y 580.304,Z 243.008,A -85,B 0,C 180,E1 -1954.92,E2 -1954.92} C_VEL
LIN {X 0,Y 580.269,Z 243.014,A -85,B 0,C 180,E1 -1957.947,E2 -1957.947} C_VEL
LIN {X 0,Y 580.313,Z 243.007,A -85,B 0,C 180,E1 -1960.913,E2 -1960.913} C_VEL
LIN {X 0,Y 580.276,Z 243.015,A -85,B 0,C 180,E1 -1963.825,E2 -1963.825} C_VEL
LIN {X 0,Y 580.319,Z 243.008,A -85,B 0,C 180,E1 -1965.982,E2 -1965.982} C_VEL
LIN {X 0,Y 580.298,Z 243.008,A -85,B 0,C 180,E1 -1968.826,E2 -1968.826} C_VEL
LIN {X 0,Y 580.328,Z 243.012,A -85,B 0,C 180,E1 -1971.643,E2 -1971.643} C_VEL
LIN {X 0,Y 580.317,Z 243.005,A -85,B 0,C 180,E1 -1974.44,E2 -1974.44} C_VEL
LIN {X 0,Y 580.338,Z 243.007,A -85,B 0,C 180,E1 -1977.223,E2 -1977.223} C_VEL
LIN {X 0,Y 580.345,Z 243.004,A -85,B 0,C 180,E1 -1979.999,E2 -1979.999} C_VEL
LIN {X 0,Y 580.34,Z 243.002,A -85,B 0,C 180,E1 -1982.776,E2 -1982.776} C_VEL
LIN {X 0,Y 580.315,Z 243.016,A -85,B 0,C 180,E1 -1985.559,E2 -1985.559} C_VEL
LIN {X 0,Y 580.328,Z 243.004,A -85,B 0,C 180,E1 -1988.355,E2 -1988.355} C_VEL
LIN {X 0,Y 580.291,Z 243.012,A -85,B 0,C 180,E1 -1991.191,E2 -1991.191} C_VEL
LIN {X 0,Y 580.317,Z 243.008,A -85,B 0,C 180,E1 -1994.016,E2 -1994.016} C_VEL
LIN {X 0,Y 580.304,Z 243.008,A -85,B 0,C 180,E1 -1996.914,E2 -1996.914} C_VEL
LIN {X 0,Y 580.298,Z 243.013,A -85,B 0,C 180,E1 -1999.822,E2 -1999.822} C_VEL
LIN {X 0,Y 580.279,Z 243.015,A -85,B 0,C 180,E1 -2001.342,E2 -2001.342} C_VEL
LIN {X 0,Y 579.581,Z 243.101,A -85,B 0,C 180,E1 -2001.921,E2 -2001.921} C_VEL
LIN {X 0,Y 576.702,Z 243.456,A -85,B 0,C 180,E1 -2002.86,E2 -2002.86} C_VEL
LIN {X 0,Y 574.307,Z 243.763,A -85,B 0,C 180,E1 -2003.617,E2 -2003.617} C_VEL
LIN {X 0,Y 573.308,Z 243.88,A -85,B 0,C 180,E1 -2004.201,E2 -2004.201} C_VEL
LIN {X 0,Y 573.242,Z 243.886,A -85,B 0,C 180,E1 -2004.398,E2 -2004.398} C_VEL
LIN {X 0,Y 573.255,Z 243.886,A -85,B 0,C 180,E1 -2006.975,E2 -2006.975} C_VEL
LIN {X 0,Y 573.241,Z 243.895,A -85,B 0,C 180,E1 -2009.489,E2 -2009.489} C_VEL
LIN {X 0,Y 573.247,Z 243.887,A -85,B 0,C 180,E1 -2012.229,E2 -2012.229} C_VEL
LIN {X 0,Y 573.245,Z 243.886,A -85,B 0,C 180,E1 -2014.774,E2 -2014.774} C_VEL
LIN {X 0,Y 573.244,Z 243.89,A -85,B 0,C 180,E1 -2017.166,E2 -2017.166} C_VEL
LIN {X 0,Y 573.238,Z 243.896,A -85,B 0,C 180,E1 -2019.607,E2 -2019.607} C_VEL
LIN {X 0,Y 573.233,Z 243.887,A -85,B 0,C 180,E1 -2022.642,E2 -2022.642} C_VEL
LIN {X 0,Y 573.229,Z 243.896,A -85,B 0,C 180,E1 -2025.667,E2 -2025.667} C_VEL
LIN {X 0,Y 573.235,Z 243.887,A -85,B 0,C 180,E1 -2028.544,E2 -2028.544} C_VEL
LIN {X 0,Y 573.239,Z 243.892,A -85,B 0,C 180,E1 -2031.299,E2 -2031.299} C_VEL
LIN {X 0,Y 573.231,Z 243.891,A -85,B 0,C 180,E1 -2034.014,E2 -2034.014} C_VEL
LIN {X 0,Y 573.275,Z 243.882,A -85,B 0,C 180,E1 -2036.519,E2 -2036.519} C_VEL
LIN {X 0,Y 573.229,Z 243.891,A -85,B 0,C 180,E1 -2039.116,E2 -2039.116} C_VEL
LIN {X 0,Y 573.256,Z 243.888,A -85,B 0,C 180,E1 -2041.968,E2 -2041.968} C_VEL
LIN {X 0,Y 573.244,Z 243.886,A -85,B 0,C 180,E1 -2044.59,E2 -2044.59} C_VEL
LIN {X 0,Y 573.247,Z 243.894,A -85,B 0,C 180,E1 -2047.663,E2 -2047.663} C_VEL
LIN {X 0,Y 573.271,Z 243.883,A -85,B 0,C 180,E1 -2050.727,E2 -2050.727} C_VEL
LIN {X 0,Y 573.249,Z 243.895,A -85,B 0,C 180,E1 -2053.622,E2 -2053.622} C_VEL
LIN {X 0,Y 573.263,Z 243.89,A -85,B 0,C 180,E1 -2055.807,E2 -2055.807} C_VEL
LIN {X 0,Y 573.274,Z 243.882,A -85,B 0,C 180,E1 -2058.734,E2 -2058.734} C_VEL
LIN {X 0,Y 573.28,Z 243.891,A -85,B 0,C 180,E1 -2061.54,E2 -2061.54} C_VEL
LIN {X 0,Y 573.275,Z 243.883,A -85,B 0,C 180,E1 -2064.372,E2 -2064.372} C_VEL
LIN {X 0,Y 573.292,Z 243.885,A -85,B 0,C 180,E1 -2067.892,E2 -2067.892} C_VEL
LIN {X 0,Y 573.318,Z 243.877,A -85,B 0,C 180,E1 -2070.702,E2 -2070.702} C_VEL
LIN {X 0,Y 573.233,Z 243.896,A -85,B 0,C 180,E1 -2073.514,E2 -2073.514} C_VEL
LIN {X 0,Y 573.278,Z 243.892,A -85,B 0,C 180,E1 -2075.628,E2 -2075.628} C_VEL
LIN {X 0,Y 573.244,Z 243.886,A -85,B 0,C 180,E1 -2078.46,E2 -2078.46} C_VEL
LIN {X 0,Y 573.261,Z 243.89,A -85,B 0,C 180,E1 -2081.312,E2 -2081.312} C_VEL
LIN {X 0,Y 573.242,Z 243.888,A -85,B 0,C 180,E1 -2084.193,E2 -2084.193} C_VEL
LIN {X 0,Y 573.246,Z 243.889,A -85,B 0,C 180,E1 -2087.111,E2 -2087.111} C_VEL
LIN {X 0,Y 573.237,Z 243.89,A -85,B 0,C 180,E1 -2090.077,E2 -2090.077} C_VEL
LIN {X 0,Y 573.22,Z 243.89,A -85,B 0,C 180,E1 -2092.338,E2 -2092.338} C_VEL
LIN {X 0,Y 573.23,Z 243.895,A -85,B 0,C 180,E1 -2095.41,E2 -2095.41} C_VEL
LIN {X 0,Y 573.235,Z 243.89,A -85,B 0,C 180,E1 -2098.028,E2 -2098.028} C_VEL
LIN {X 0,Y 573.215,Z 243.891,A -85,B 0,C 180,E1 -2100.882,E2 -2100.882} C_VEL
LIN {X 0,Y 573.233,Z 243.892,A -85,B 0,C 180,E1 -2103.168,E2 -2103.168} C_VEL
LIN {X 0,Y 573.08,Z 256.108,A -85,B 0,C 180,E1 -2106.06,E2 -2106.06} C_VEL
LIN {X 0,Y 573.034,Z 265.158,A -85,B 0,C 180,E1 -2108.183,E2 -2108.183} C_VEL
LIN {X 0,Y 573.632,Z 270.665,A -85,B 0,C 180,E1 -2108.277,E2 -2108.277} C_VEL
LIN {X 0,Y 573.493,Z 340.066,A -85,B 0,C 180,E1 -2109.16,E2 -2109.16} C_VEL
LIN {X 0,Y 573.421,Z 350.102,A -85,B 0,C 180,E1 -2109.388,E2 -2109.388} C_VEL
LIN {X 0,Y 573.348,Z 361.179,A -85,B 0,C 180,E1 -2109.769,E2 -2109.769} C_VEL
LIN {X 0,Y 573.302,Z 371.706,A -85,B 0,C 180,E1 -2110.288,E2 -2110.288} C_VEL
LIN {X 0,Y 573.286,Z 379.149,A -85,B 0,C 180,E1 -2110.751,E2 -2110.751} C_VEL
LIN {X 0,Y 573.201,Z 386.907,A -85,B 0,C 180,E1 -2111.341,E2 -2111.341} C_VEL
LIN {X 0,Y 573.17,Z 393.742,A -85,B 0,C 180,E1 -2111.971,E2 -2111.971} C_VEL
LIN {X 0,Y 573.085,Z 399.698,A -85,B 0,C 180,E1 -2112.626,E2 -2112.626} C_VEL
LIN {X 0,Y 573.061,Z 405.341,A -85,B 0,C 180,E1 -2113.375,E2 -2113.375} C_VEL
LIN {X 0,Y 573.054,Z 410.208,A -85,B 0,C 180,E1 -2114.161,E2 -2114.161} C_VEL
LIN {X 0,Y 572.995,Z 414.494,A -85,B 0,C 180,E1 -2115.025,E2 -2115.025} C_VEL
LIN {X 0,Y 572.989,Z 418.264,A -85,B 0,C 180,E1 -2116.027,E2 -2116.027} C_VEL
LIN {X 0,Y 572.961,Z 419.947,A -85,B 0,C 180,E1 -2116.616,E2 -2116.616} C_VEL
LIN {X 0,Y 572.975,Z 421.848,A -85,B 0,C 180,E1 -2117.577,E2 -2117.577} C_VEL
LIN {X 0,Y 572.937,Z 422.79,A -85,B 0,C 180,E1 -2118.518,E2 -2118.518} C_VEL
LIN {X 0,Y 572.931,Z 422.818,A -85,B 0,C 180,E1 -2119.51,E2 -2119.51} C_VEL
LIN {X 0,Y 572.935,Z 421.724,A -85,B 0,C 180,E1 -2120.604,E2 -2120.604} C_VEL
LIN {X 0,Y 572.982,Z 419.359,A -85,B 0,C 180,E1 -2121.719,E2 -2121.719} C_VEL
LIN {X 0,Y 573.003,Z 415.354,A -85,B 0,C 180,E1 -2122.865,E2 -2122.865} C_VEL
LIN {X 0,Y 573.024,Z 411.354,A -85,B 0,C 180,E1 -2123.718,E2 -2123.718} C_VEL
LIN {X 0,Y 573.059,Z 407.282,A -85,B 0,C 180,E1 -2124.424,E2 -2124.424} C_VEL
LIN {X 0,Y 573.106,Z 401.451,A -85,B 0,C 180,E1 -2125.245,E2 -2125.245} C_VEL
LIN {X 0,Y 573.138,Z 395.061,A -85,B 0,C 180,E1 -2125.982,E2 -2125.982} C_VEL
LIN {X 0,Y 573.187,Z 388.404,A -85,B 0,C 180,E1 -2126.619,E2 -2126.619} C_VEL
LIN {X 0,Y 573.265,Z 381.795,A -85,B 0,C 180,E1 -2127.148,E2 -2127.148} C_VEL
LIN {X 0,Y 573.351,Z 373.907,A -85,B 0,C 180,E1 -2127.671,E2 -2127.671} C_VEL
LIN {X 0,Y 573.347,Z 365.592,A -85,B 0,C 180,E1 -2128.116,E2 -2128.116} C_VEL
LIN {X 0,Y 573.4,Z 356.221,A -85,B 0,C 180,E1 -2128.505,E2 -2128.505} C_VEL
LIN {X 0,Y 573.498,Z 344.69,A -85,B 0,C 180,E1 -2128.845,E2 -2128.845} C_VEL
LIN {X 0,Y 573.523,Z 328.859,A -85,B 0,C 180,E1 -2129.09,E2 -2129.09} C_VEL
LIN {X 0,Y 573.541,Z 268.513,A -85,B 0,C 180,E1 -2129.842,E2 -2129.842} C_VEL
LIN {X 0,Y 573.087,Z 265.126,A -85,B 0,C 180,E1 -2129.914,E2 -2129.914} C_VEL
LIN {X 0,Y 573.152,Z 253.577,A -85,B 0,C 180,E1 -2132.625,E2 -2132.625} C_VEL
LIN {X 0,Y 573.253,Z 243.889,A -85,B 0,C 180,E1 -2134.967,E2 -2134.967} C_VEL
LIN {X 0,Y 573.228,Z 243.889,A -85,B 0,C 180,E1 -2137.663,E2 -2137.663} C_VEL
LIN {X 0,Y 573.246,Z 243.889,A -85,B 0,C 180,E1 -2139.924,E2 -2139.924} C_VEL
LIN {X 0,Y 573.252,Z 243.888,A -85,B 0,C 180,E1 -2142.989,E2 -2142.989} C_VEL
LIN {X 0,Y 573.261,Z 243.885,A -85,B 0,C 180,E1 -2145.807,E2 -2145.807} C_VEL
LIN {X 0,Y 573.272,Z 243.889,A -85,B 0,C 180,E1 -2148.734,E2 -2148.734} C_VEL
LIN {X 0,Y 573.297,Z 243.88,A -85,B 0,C 180,E1 -2151.541,E2 -2151.541} C_VEL
LIN {X 0,Y 573.284,Z 243.89,A -85,B 0,C 180,E1 -2154.372,E2 -2154.372} C_VEL
LIN {X 0,Y 573.3,Z 243.88,A -85,B 0,C 180,E1 -2157.893,E2 -2157.893} C_VEL
LIN {X 0,Y 573.328,Z 243.882,A -85,B 0,C 180,E1 -2160.703,E2 -2160.703} C_VEL
LIN {X 0,Y 573.232,Z 243.887,A -85,B 0,C 180,E1 -2163.515,E2 -2163.515} C_VEL
LIN {X 0,Y 573.284,Z 243.881,A -85,B 0,C 180,E1 -2165.629,E2 -2165.629} C_VEL
LIN {X 0,Y 573.298,Z 243.888,A -85,B 0,C 180,E1 -2168.46,E2 -2168.46} C_VEL
LIN {X 0,Y 573.262,Z 243.884,A -85,B 0,C 180,E1 -2171.313,E2 -2171.313} C_VEL
LIN {X 0,Y 573.264,Z 243.888,A -85,B 0,C 180,E1 -2174.194,E2 -2174.194} C_VEL
LIN {X 0,Y 573.251,Z 243.886,A -85,B 0,C 180,E1 -2177.112,E2 -2177.112} C_VEL
LIN {X 0,Y 573.249,Z 243.889,A -85,B 0,C 180,E1 -2180.077,E2 -2180.077} C_VEL
LIN {X 0,Y 573.23,Z 243.894,A -85,B 0,C 180,E1 -2182.338,E2 -2182.338} C_VEL
LIN {X 0,Y 573.251,Z 243.884,A -85,B 0,C 180,E1 -2185.411,E2 -2185.411} C_VEL
LIN {X 0,Y 573.258,Z 243.887,A -85,B 0,C 180,E1 -2188.033,E2 -2188.033} C_VEL
LIN {X 0,Y 573.229,Z 243.892,A -85,B 0,C 180,E1 -2190.884,E2 -2190.884} C_VEL
LIN {X 0,Y 573.255,Z 243.883,A -85,B 0,C 180,E1 -2193.525,E2 -2193.525} C_VEL
LIN {X 0,Y 573.255,Z 243.888,A -85,B 0,C 180,E1 -2196.049,E2 -2196.049} C_VEL
LIN {X 0,Y 573.242,Z 243.893,A -85,B 0,C 180,E1 -2198.702,E2 -2198.702} C_VEL
LIN {X 0,Y 573.237,Z 243.887,A -85,B 0,C 180,E1 -2201.595,E2 -2201.595} C_VEL
LIN {X 0,Y 573.23,Z 243.895,A -85,B 0,C 180,E1 -2204.334,E2 -2204.334} C_VEL
LIN {X 0,Y 573.235,Z 243.887,A -85,B 0,C 180,E1 -2207.359,E2 -2207.359} C_VEL
LIN {X 0,Y 573.235,Z 243.896,A -85,B 0,C 180,E1 -2210.393,E2 -2210.393} C_VEL
LIN {X 0,Y 573.251,Z 243.887,A -85,B 0,C 180,E1 -2213.079,E2 -2213.079} C_VEL
LIN {X 0,Y 573.263,Z 243.884,A -85,B 0,C 180,E1 -2215.672,E2 -2215.672} C_VEL
LIN {X 0,Y 573.238,Z 243.892,A -85,B 0,C 180,E1 -2218.185,E2 -2218.185} C_VEL
LIN {X 0,Y 573.258,Z 243.893,A -85,B 0,C 180,E1 -2220.635,E2 -2220.635} C_VEL
LIN {X 0,Y 573.229,Z 243.888,A -85,B 0,C 180,E1 -2223.51,E2 -2223.51} C_VEL
LIN {X 0,Y 573.231,Z 243.893,A -85,B 0,C 180,E1 -2226.135,E2 -2226.135} C_VEL
LIN {X 0,Y 573.276,Z 244.089,A -85,B 0,C 180,E1 -2227.141,E2 -2227.141} C_VEL
LIN {X 0,Y 573.801,Z 248.851,A -85,B 0,C 180,E1 -2227.876,E2 -2227.876} C_VEL
LIN {X 0,Y 573.702,Z 263.63,A -85,B 0,C 180,E1 -2230.127,E2 -2230.127} C_VEL
LIN {X 0,Y 573.503,Z 280.312,A -85,B 0,C 180,E1 -2232.713,E2 -2232.713} C_VEL
LIN {X 0,Y 573.379,Z 298.709,A -85,B 0,C 180,E1 -2235.539,E2 -2235.539} C_VEL
LIN {X 0,Y 573.242,Z 317.103,A -85,B 0,C 180,E1 -2238.329,E2 -2238.329} C_VEL
LIN {X 0,Y 573.168,Z 322.309,A -85,B 0,C 180,E1 -2239.113,E2 -2239.113} C_VEL
LIN {X 0,Y 573.641,Z 328.425,A -85,B 0,C 180,E1 -2239.204,E2 -2239.204} C_VEL
LIN {X 0,Y 573.56,Z 399.161,A -85,B 0,C 180,E1 -2240.1,E2 -2240.1} C_VEL
LIN {X 0,Y 573.475,Z 408.426,A -85,B 0,C 180,E1 -2240.299,E2 -2240.299} C_VEL
LIN {X 0,Y 573.421,Z 416.899,A -85,B 0,C 180,E1 -2240.565,E2 -2240.565} C_VEL
LIN {X 0,Y 573.364,Z 425.405,A -85,B 0,C 180,E1 -2240.92,E2 -2240.92} C_VEL
LIN {X 0,Y 573.333,Z 433.735,A -85,B 0,C 180,E1 -2241.364,E2 -2241.364} C_VEL
LIN {X 0,Y 573.253,Z 441.774,A -85,B 0,C 180,E1 -2241.895,E2 -2241.895} C_VEL
LIN {X 0,Y 573.175,Z 450.435,A -85,B 0,C 180,E1 -2242.603,E2 -2242.603} C_VEL
LIN {X 0,Y 573.159,Z 458.429,A -85,B 0,C 180,E1 -2243.424,E2 -2243.424} C_VEL
LIN {X 0,Y 573.113,Z 464.436,A -85,B 0,C 180,E1 -2244.194,E2 -2244.194} C_VEL
LIN {X 0,Y 572.995,Z 469.989,A -85,B 0,C 180,E1 -2245.075,E2 -2245.075} C_VEL
LIN {X 0,Y 573.037,Z 475.149,A -85,B 0,C 180,E1 -2246.132,E2 -2246.132} C_VEL
LIN {X 0,Y 572.99,Z 477.789,A -85,B 0,C 180,E1 -2246.836,E2 -2246.836} C_VEL
LIN {X 0,Y 572.94,Z 480.682,A -85,B 0,C 180,E1 -2247.891,E2 -2247.891} C_VEL
LIN {X 0,Y 572.944,Z 481.935,A -85,B 0,C 180,E1 -2248.594,E2 -2248.594} C_VEL
LIN {X 0,Y 572.937,Z 482.71,A -85,B 0,C 180,E1 -2249.297,E2 -2249.297} C_VEL
LIN {X 0,Y 572.935,Z 483,A -85,B 0,C 180,E1 -2250,E2 -2250} C_VEL
LIN {X 0,Y 572.937,Z 482.709,A -85,B 0,C 180,E1 -2250.703,E2 -2250.703} C_VEL
LIN {X 0,Y 572.944,Z 481.934,A -85,B 0,C 180,E1 -2251.406,E2 -2251.406} C_VEL
LIN {X 0,Y 572.94,Z 480.681,A -85,B 0,C 180,E1 -2252.109,E2 -2252.109} C_VEL
LIN {X 0,Y 572.99,Z 477.787,A -85,B 0,C 180,E1 -2253.164,E2 -2253.164} C_VEL
LIN {X 0,Y 573.037,Z 475.148,A -85,B 0,C 180,E1 -2253.868,E2 -2253.868} C_VEL
LIN {X 0,Y 572.995,Z 469.985,A -85,B 0,C 180,E1 -2254.925,E2 -2254.925} C_VEL
